(* CODESYS project cy-09-ifm-022_003.project
   Title: cy-09-ifm
   Author: AR
   Company: Clevergy S.r.l

Project tree, tasks and I/O mapping:
  Device : AC14nn, ifm electronic, order no. AC14nn, version 3.5.3.002
    application Application
      libraries: Standard, 3.5.5.0 (System); ACnnnn_Utils, * (ifm electronic); Util, 3.5.1.0 (System); SysRtc23, 3.4.0.0 (System); SysSocket23, 3.5.4.10 (System); SysFile, 3.5.6.0 (System); SysTypes Interfaces, * (System); CmpErrors Interfaces, * (System); VisuDialogs, * (System); NETWORK, 1.2.1.0 (OSCAT)
      task MainTask (cyclic, interval t#20ms, priority 15) calls PLC_PRG
      task EventTask (cyclic, interval t#20ms, priority 5) calls PLC_RT
      task VISU_TASK (cyclic, interval 100 ms, priority 30) calls VisuElems.Visu_Prg
      visualisation VIS_CHONOEDITOR
      visualisation PLC_VISU
    ASi_Master_1 : ASi Master 1, ifm electronic, version 3.5.3.002
      ASi_1_binaryIO : ASi_1_binaryIO, ifm ecomatic gmbh, version 3.5.3.002
          input  PSG01_IN : BOOL  // ASi Input bin.Digital S(A) Slave.Digital S(A) Slave[1].Bit0
          input  PSG02_IN : BOOL  // ASi Input bin.Digital S(A) Slave.Digital S(A) Slave[1].Bit2
          input  EXT_KEY1 : BOOL  // ASi Input bin.Digital S(A) Slave.Digital S(A) Slave[1].Bit3
          input  PSG03_IN : BOOL  // ASi Input bin.Digital S(A) Slave.Digital S(A) Slave[2].Bit0
          input  PSG04_IN : BOOL  // ASi Input bin.Digital S(A) Slave.Digital S(A) Slave[2].Bit2
          input  PSG05_IN : BOOL  // ASi Input bin.Digital S(A) Slave.Digital S(A) Slave[3].Bit0
          input  PSG06_IN : BOOL  // ASi Input bin.Digital S(A) Slave.Digital S(A) Slave[3].Bit2
          input  PSG07_IN : BOOL  // ASi Input bin.Digital S(A) Slave.Digital S(A) Slave[4].Bit0
          input  PSG08_IN : BOOL  // ASi Input bin.Digital S(A) Slave.Digital S(A) Slave[4].Bit2
          input  PSG09_IN : BOOL  // ASi Input bin.Digital S(A) Slave.Digital S(A) Slave[5].Bit0
          input  PSG10_IN : BOOL  // ASi Input bin.Digital S(A) Slave.Digital S(A) Slave[5].Bit2
          input  EXT_KEY2 : BOOL  // ASi Input bin.Digital S(A) Slave.Digital S(A) Slave[5].Bit3
          input  PSG11_IN : BOOL  // ASi Input bin.Digital S(A) Slave.Digital S(A) Slave[6].Bit0
          input  PSG12_IN : BOOL  // ASi Input bin.Digital S(A) Slave.Digital S(A) Slave[6].Bit2
          input  PSG13_IN : BOOL  // ASi Input bin.Digital S(A) Slave.Digital S(A) Slave[7].Bit0
          input  EXT_KEY3 : BOOL  // ASi Input bin.Digital S(A) Slave.Digital S(A) Slave[7].Bit3
          input  PSG14_IN : BOOL  // ASi Input bin.Digital S(A) Slave.Digital S(A) Slave[8].Bit0
          input  PSG15_IN : BOOL  // ASi Input bin.Digital S(A) Slave.Digital S(A) Slave[8].Bit2
          input  PSG16_IN : BOOL  // ASi Input bin.Digital S(A) Slave.Digital S(A) Slave[9].Bit0
          input  PSG17_IN : BOOL  // ASi Input bin.Digital S(A) Slave.Digital S(A) Slave[9].Bit2
          unmapped channels: ASi Input bin, ASi Output bin
      ASi_1_analogIO : ASi_1_analogIO, ifm ecomatic gmbh, version 3.5.3.002
          unmapped channels: ASi Input, ASi Output
    ASi_Master_2 : ASi Master 2, ifm electronic, version 3.5.3.002
      ASi_2_binaryIO : ASi_2_binaryIO, ifm ecomatic gmbh, version 3.5.3.002
          input  PSG18_IN : BOOL  // ASi Input bin.Digital S(A) Slave.Digital S(A) Slave[10].Bit0
          input  PSG19_IN : BOOL  // ASi Input bin.Digital S(A) Slave.Digital S(A) Slave[10].Bit2
          input  PSG20_IN : BOOL  // ASi Input bin.Digital S(A) Slave.Digital S(A) Slave[11].Bit0
          input  PSG21_IN : BOOL  // ASi Input bin.Digital S(A) Slave.Digital S(A) Slave[11].Bit1
          input  PSG22_IN : BOOL  // ASi Input bin.Digital S(A) Slave.Digital S(A) Slave[11].Bit2
          input  PSG23_IN : BOOL  // ASi Input bin.Digital S(A) Slave.Digital S(A) Slave[12].Bit0
          input  PSG24_IN : BOOL  // ASi Input bin.Digital S(A) Slave.Digital S(A) Slave[13].Bit0
          input  PSG25_IN : BOOL  // ASi Input bin.Digital S(A) Slave.Digital S(A) Slave[13].Bit1
          input  PSG26_IN : BOOL  // ASi Input bin.Digital S(A) Slave.Digital S(A) Slave[13].Bit2
          input  PSG27_IN : BOOL  // ASi Input bin.Digital S(A) Slave.Digital S(A) Slave[14].Bit0
          input  PSG28_IN : BOOL  // ASi Input bin.Digital S(A) Slave.Digital S(A) Slave[14].Bit1
          input  PSG29_IN : BOOL  // ASi Input bin.Digital S(A) Slave.Digital S(A) Slave[14].Bit2
          input  PSG30_IN : BOOL  // ASi Input bin.Digital S(A) Slave.Digital S(A) Slave[15].Bit0
          input  PSG31_IN : BOOL  // ASi Input bin.Digital S(A) Slave.Digital S(A) Slave[15].Bit1
          input  PSG32_IN : BOOL  // ASi Input bin.Digital S(A) Slave.Digital S(A) Slave[15].Bit2
          input  PSG33_IN : BOOL  // ASi Input bin.Digital S(A) Slave.Digital S(A) Slave[16].Bit0
          input  PSG34_IN : BOOL  // ASi Input bin.Digital S(A) Slave.Digital S(A) Slave[17].Bit0
          unmapped channels: ASi Input bin, ASi Output bin
      ASi_2_analogIO : ASi_2_analogIO, ifm ecomatic gmbh, version 3.5.3.002
          unmapped channels: ASi Input, ASi Output
    Fieldbus_Interface : Fieldbus Interface, ifm electronic, version 3.5.3.002
      FieldBusData_ : FieldBusData  , ifm ecomatic gmbh, version 3.5.3.002
          unmapped channels: Inputs from fieldbus, Outputs to fieldbus
      ASi_1_binaryOut : ASi_1_binaryOut, ifm ecomatic gmbh, version 3.5.3.002
          unmapped channels: FB ASi Output bin
      ASi_1_analogOut : ASi_1_analogOut, ifm ecomatic gmbh, version 3.5.3.002
          unmapped channels: FB ASi Output ana
      ASi_2_binaryOut : ASi_2_binaryOut, ifm ecomatic gmbh, version 3.5.3.002
          unmapped channels: FB ASi Output bin
      ASi_2_analogOut : ASi_2_analogOut, ifm ecomatic gmbh, version 3.5.3.002
          unmapped channels: FB ASi Output ana
    Ethernet : Ethernet, ifm electronic, version 3.4.2.0
        settings: IPAddress = [192,168,100,2]; SubnetMask = [255,255,255,0]; GatewayAddress = [0,0,0,0]
  POUs/
    Utils Functions/
      function ADDSTRING [ST]
      function block AVERAGE_DINT [ST]: Read, Reset
      function block AVERAGE_INT [ST]: Read, Reset
      function block AVERAGE_T [ST]: Read, Reset
      function CHKSTRING [ST]
      function COPY_32SWAP16 [ST]
      function DWORDSWAP [ST]
      function block FLT_EVENT [ST]
      function block FLT_TAP [ST]
      function block FLT_TIME [ST]
      function HEXTORAW [ST]
      function LINEAR [ST]
      function LINEAR_BAD [ST]
      function MEMCLR [ST]
      function MEMCPY [ST]
      function block DELAYRETRY [ST]: Start, Success, Fail
      function RAW16TOHEXSTR [ST]
      function RAWTOHEX [ST]
      function RAWTOHEXSTR [ST]
      function STR_NOSPACES [ST]
      function block TCPCLIENT [ST]
      function block TCPSERVER [ST]
      function block TONOF [ST]
      function ADR_AT_INT [ST]
    Utils/
      function CSV_Log [ST]
      function RTC_Update [ST]
    TCP_Logger/
      function LogEv [ST]
      function Logger_Head [ST]
      program Logger_Proc [ST]: MsgChk, MsgSave
      function Logger_Send [ST]
      function LogTrig [ST]
    Plant_Objects/
      function block obj_LUXM [ST]: AddLogData, StatReset
      function block obj_ZREL [ST]: AddLogData, MB_Req_NetStatus, MB_Set_DefaultMode, MB_Req_Status, MB_Set_AutoLearn, MB_Response
      function block obj_CRON [ST]: DB_Create, DB_Load, DB_SetName, Init, AddLogData
      function block obj_CRON_EDITOR [ST]: CA_Load_Exe, CA_Save_Exe, FileOpen, JL_Load_Exe, JL_Save_Exe, PR_Load_Exe, PR_Save_Exe
      function block obj_MODBUS_TCP [ST]: VARS_Process, VAR_Search
      function block obj_ASI [ST]
      function block obj_PSG [ST]: StatReset, AddLogData
      function block obj_ZGW [ST]: AddLogData
      function block obj_LICENSE [ST]
    program PLC_PRG [ST]: Main_Stm
    TCP_Remote/
      program Remote_Proc [ST]: Cmd_CAL, Cmd_CRON, Cmd_GRU, Cmd_PDC, Cmd_SYS, Command, Cmd_LUX
    Plant/
    program PLC_RT [ST]
    WagoLibModbus_IP_01/
      function block Client_OpenClose [ST]
      function block ETHERNET_MODBUSMASTER_TCP [ST]
      function Modbus_IP_Version [ST]
      function ModbusRequest [ST]
  _Datatypes/
    Logger/
      data type en_Logger_ErrLev
      data type en_Logger_Status
      data type typ_Logger
    data type en_SYS_Objects
    data type en_SYS_Status
    data type typ_SYS
    WagoLibModbus_IP_1/
      data type MODBUS_FC
    Plant_Objects/
      data type typ_Cron_Calendar
      data type typ_Cron_Jolly
      data type typ_Cron_Profile
      data type typ_MODBUS_VAR
  _Variables/
    global variables Global_Constants
    global variables Global_Retain
    global variables Global_Variables
  text list GlobalTextList
*)

// _Datatypes/Logger/en_Logger_ErrLev
TYPE en_Logger_ErrLev :
(
	EL_Log			:=0,
	EL_Wrn			:=1,
	EL_Alarm		:=2,
	EL_AlarmStop	:=3
);
END_TYPE

// _Datatypes/Logger/en_Logger_Status
TYPE en_Logger_Status :
(
	S_Logger_UNKNOWN := 0,
	S_Logger_IDLE,
	S_Logger_WAITCONN,
	S_Logger_WAITTX,
	S_Logger_WAITRESP,
	S_Logger_ERROR
);
END_TYPE

// _Datatypes/en_SYS_Objects
TYPE en_SYS_Objects :
(
	EO_SYS		:=0,  (* PLC *)
	EO_VPN		:=1,  (* VPN *)
	EO_DOOR		:=2,  (* Door & access control *)

	EO_CAL		:=10, (* Caldaia *)
	EO_CIR		:=11, (* Circolatore *)
	EO_CRON		:=12, (* Crono-termostato *)
	EO_VRD		:=13, (* Valvola miscelatore pannelli *)
	EO_CTL		:=14, (* Contalitri *)
	EO_CTB		:=15, (* Contabilizzatore *)
	EO_TPV		:=16, (* Temperature probes values *)
	EO_PPV		:=17, (* Pressure probes values *)
	EO_PBV		:=18, (* Over-Pressure Alarms *)
	EO_TBV		:=19, (* Over-Temperature Alarms *)
	EO_PMV		:=20, (* Under-Pressure Alarms *)
	EO_GRU		:=21, (* Gruppo termico *)
	EO_PDC		:=22, (* Pompa di calore *)
	EO_SOL		:=23, (* Pannello solare termico *)
	EO_ESOL		:=24, (* Pannello solare fotovoltaico *)
	EO_GAS		:=25, (* Contatore GAS *)
	EO_PORT		:=26, (* Misuratore di portata *)
	EO_FPV		:=27, (* Flow probes values *)
	EO_ANZ		:=28, (* Analizzatore di rete *)
	EO_SCA		:=29, (* Signal Control Alarms *)
	EO_LUX		:=30, (* Base Illumination point *)
	EO_LUXM		:=31, (* Metered Illumination point *)
	EO_PSG		:=32, (* Sensore di passaggio *)
	EO_HVAC		:=33, (* Heating, Ventilating and Air Conditioning *)
	EO_HYGRV	:=34, (* Relative Humidity sensors value *)
	EO_COOV		:=35, (* Carbon Dioxide CO2 sensors value *)

	EO_ZGW			:=200,  (* ZigBee - Gateway *)
	EO_ZRM			:=201,	(* ZigBee - Repeater *)
	EO_ZREL			:=202,	(* ZigBee - Actuator rele *)
	EO_ZTHL			:=203,	(* ZigBee - Temperature Sensor *)

	EO_ASGW			:=250,	(* ASi - Gateway *)
	EO_ASCBI		:=251,	(* ASi - Input Board, Ciabatta *)

	EO_LON			:=1000, (* Bus - LON *)
	EO_MODBUS		:=1001, (* Bus - MODBUS *)
	EO_MBUS			:=1002, (* Bus - M-BUS *)
	EO_MODBUS_TCP	:=1003, (* Bus - MODBUS TCP *)

	EO_GENERIC		:=9000, (* Generic dataset *)
	EO_EXPO			:=9001  (* EXPO dataset *)
);
END_TYPE

// _Datatypes/en_SYS_Status
TYPE en_SYS_Status :
(
	S_UNKNOWN  := 0,
	S_STARTUP,
	S_INIT_RTC,
	S_INIT_VAR,
	S_AUTOTEST,
	S_RUNNING,
	S_SHUTDOWN,
	S_HALT
);
END_TYPE

// _Datatypes/Logger/typ_Logger
TYPE typ_Logger :
STRUCT
	Status		: en_Logger_Status;

	SendReq		: BOOL;
	SendIdx		: DWORD;
	SendData	: ARRAY [0..MAX_SEND_TCP_CLIENT] OF BYTE;
	SendLen		: DINT;

	TData		: ARRAY [0..MAX_SEND_TCP_CLIENT] OF BYTE;
	TLen		: DINT;

	LastIdxPos	: DWORD;

	(* Temporary variables used by objects *)
	s1			: STRING(256);
	i1			: WORD;

END_STRUCT
END_TYPE

// _Datatypes/typ_SYS
TYPE typ_SYS :
STRUCT
	Status			: en_SYS_Status;
	Warning			: BOOL;
	Alarm			: BOOL;
	AlarmStop		: BOOL;

	Time_LogString	: STRING;
	Time_Year		: WORD;
	Time_Month		: BYTE;
	Time_Day		: BYTE;

	Time_CT_DT		: DT;
	Time_CT_Day		: WORD;
	Time_CT_Quarter	: BYTE;

	LastLogs_Idx	: BYTE;
	LastLogs_Dat	: ARRAY[0..5] OF STRING;
	LastLogs_Msg	: ARRAY[0..5] OF STRING;

END_STRUCT
END_TYPE

// _Datatypes/Plant_Objects/typ_Cron_Calendar
TYPE typ_Cron_Calendar :
STRUCT
	Profile		: ARRAY[0..384] OF BYTE;
END_STRUCT
END_TYPE

// _Datatypes/Plant_Objects/typ_Cron_Jolly
TYPE typ_Cron_Jolly :
STRUCT
	Start		: DT;
	End			: DT;
	Temp		: INT;
	Flags		: WORD; (* B0:Enabled B1..B15:Unused *)
END_STRUCT
END_TYPE

// _Datatypes/Plant_Objects/typ_Cron_Profile
TYPE typ_Cron_Profile :
STRUCT
	Flags		: WORD;
	Setpoint	: ARRAY [0..95] OF INT;
END_STRUCT
END_TYPE

// _Datatypes/Plant_Objects/typ_MODBUS_VAR
TYPE typ_MODBUS_VAR : (* Gestione parametri MODBUS *)
STRUCT
	SlaveAddress	: BYTE;
	FunCode			: BYTE;
	FunAddress		: WORD;
	Refresh_Time	: BYTE; (* 0:No refresh, x:Refresh in seconds *)
	Refresh_Cnt		: BYTE; (* -- INTERNAL do not use! -- *)
	Variable		: POINTER TO ARRAY[0..99] OF WORD;
	Variable_Size	: WORD; (* 1-100:Standard reading, 1001-1100:Swap32 *)
	Variable_Mirror : WORD; (* CHECKSUM - INTERNAL [Force refresh on read variables when <>0] *)
END_STRUCT
END_TYPE

// _Datatypes/WagoLibModbus_IP_1/MODBUS_FC
TYPE MODBUS_FC : (
	(*
	 * Class 0
 	*)
	READ_MULTIPLE_REGISTERS		:=16#03,
	WRITE_MULTIPLE_REGISTERS	:=16#10,
	(*
	 * Class 1
	 *)
	READ_COILS					:=16#01,
	READ_INPUT_DISCRETES		:=16#02,
	READ_INPUT_REGISTERS		:=16#04,
	WRITE_COIL					:=16#05,
	WRITE_SINGLE_REGISTER		:=16#06,
	READ_EXCEPTION_STATUS		:=16#07,
	(*
	 * Class 2
	 *)
	FORCE_MULTIPLE_COILS		:=16#0F,
	READ_WRITE_REGISTERS		:=16#17,

	(*
	 * Class ??
	 *)
	WRITE_MASK_REGISTER			:=16#16 (* 02.04.2013 UU *)

	);
END_TYPE

// _Variables/Global_Constants
{attribute 'global_init_slot' := '300'}
VAR_GLOBAL CONSTANT

	PSG_MAX	 : BYTE := 34;
	ZREL_MAX : BYTE := 38;
	CRON_MAX : BYTE := 38;
	LUXM_MAX : BYTE := 38;
	ACTIVELUX: BYTE := 17;

	(* Filesystem *)
	LogsPath			: STRING :='/media/sd/';
	ConfPath			: STRING :='/media/sd/';
	//FilesPath			: STRING :='/media/sd/';(*'';*)(*'S:\';*)

	(* Visu colours *)	
	COLOR_RED 		: DWORD:=16#F02020;
	COLOR_YELLOW	: DWORD:=16#F0F020;
	COLOR_GREEN		: DWORD:=16#20F020;
	COLOR_GREEN_OFF : DWORD:=16#108010;
	COLOR_LBLUE		: DWORD:=16#80F0F0;
	COLOR_GREY		: DWORD:=16#C0C0C0;
	
	(******************************************************)
	(**************** MOVE OUTSIDE HERE *******************)
	(* TCP Logger *)
	Logger_SERVER		: STRING:='';
	Logger_IP			: STRING:='192.168.100.3'; //'192.168.100.3';   '178.33.227.41';
	Logger_PORT			: WORD  :=80;
	Logger_GETSTART		: STRING:='GET /cygmsrv/AFLgm.ashx?';
	Logger_GETEND		: STRING:='$R$N$R$N';
	Logger_CHECK		: STRING:='True';
	Logger_CRLF			: STRING:='$R$N';
	Logger_DataFile		: STRING:='LOG.DAT';
	Logger_DataFileOld	: STRING:='LOG.BCK';
	Logger_IndexFile	: STRING:='LOG.IDX';
	Logger_ConnRetries	: BYTE:=5;
	Logger_RecoverMsgs	: BYTE:=50;
	(* TCP Remote *)
	Remote_PORT			: WORD  :=10;
	Remote_WELCOME		: STRING:='Connected$R$N';
	(* TCP Sockets *)
	MAX_SEND_TCP_SERVER					 : DWORD:=1500;(*60000*)
	MAX_RECEIVE_TCP_SERVER				 : WORD:=3000;	//DWORD:=3000; GIURE ver 22_001
	MAX_RECEIVE_TCP_SERVER_SOCKET	 	 : DWORD:=1500;
	MAX_SEND_TCP_CLIENT					 : DWORD:=4096;(*15000*)
	MAX_RECEIVE_TCP_CLIENT				 : DWORD:=1500;
	MAX_RECEIVE_TCP_CLIENT_SOCKET		 : DWORD:=1500;
	MAX_RECEIVE_UDP_SERVER				 : INT  :=1472;
	MAX_RECEIVE_UDP_CLIENT				 : INT  :=1472;
	CONNECT_WATCHDOG_TIME				 : TIME :=T#10S;
	(******************************************************)

END_VAR

// _Variables/Global_Retain
VAR_GLOBAL RETAIN
	Mode_Manual : BOOL := FALSE;

	PASSAGES		: ARRAY [1..PSG_MAX] OF DWORD;

	WORKINGTIME		: ARRAY [1..LUXM_MAX] OF DWORD; (* [sec] Internal working time counter *)
	POWERONCYCLES	: ARRAY [1..LUXM_MAX] OF DWORD; (* Internal counter of power-on cycles *)
	ENERGYCOUNTER	: ARRAY [1..LUXM_MAX] OF DWORD; (* [E-1 kWh] Internal energy counter *)
	ENERGYCOUNTER_T : ARRAY [1..LUXM_MAX] OF DWORD; (* Temporary energy in E-2*Wsec *)
	
	LicenseManager:obj_LICENSE;

END_VAR

// _Variables/Global_Variables
VAR_GLOBAL
	Plant_NAME			: STRING :='cySN:9 cyVER:18 - AF-Logistics Bazar';	//'cySN:9 cyVER:18 - AF-Logistics Bazar';	
	Plant_SN			: DWORD  :=9;	//:=9; 	(* S/N Impianto di telecontrollo *)
	Plant_SW_VER		: WORD   :=18;		(* Versione SW installata *)

	SYS    : typ_SYS;
	Logger : typ_Logger;
	CronEd : obj_CRON_EDITOR;

	(**** PLANT OBJECTS ****)
	ASI01: obj_ASI				:=( ID:=1 );
	ASI02: obj_ASI				:=( ID:=2 );

	PSG		: ARRAY [1..PSG_MAX] OF obj_PSG;
	
	MODB01 : obj_MODBUS_TCP		:= ( ID:=1, IP:='192.168.100.4');	//'192.168.100.4' ); '10.186.79.9'
	ZGW01  : obj_ZGW			:= ( ID:=1, ADDRESS:=99  );

	ZREL   : ARRAY [1..ZREL_MAX] OF obj_ZREL;
	CRON   : ARRAY [1..CRON_MAX] OF obj_CRON;
	LUXM   : ARRAY [1..LUXM_MAX] OF obj_LUXM;
	
	ZREL_STATUS_ALIGNED   : ARRAY [1..ZREL_MAX] OF BOOL;

	(**** SIMULATION ONLY ****)
	TEST1:BOOL;	
	KEYON:BOOL;
	KEYVIRT:BOOL;
	(*...*)
	
	testCronoOn:BOOL:=FALSE;
	testCronoOff:BOOL:=FALSE;

END_VAR

// POUs/PLC_PRG
PROGRAM PLC_PRG
VAR
	Timer1	: TON; (* Fast controls tick *)
	Timer2	: TON; (* Plant control tick *)
	Timer3	: TON; (* Logger timer *)
	i 		: BYTE;
	ValInCrono	:	INT; //Valore del setpoint del crono
	LuxSelected	:	INT;//lux selezionato in plc visu per on/off
	TimerLuxSelected	:	INT;//lux selezionato in plc visu per modifica timer
	//ListaLux 	:	ARRAY [ACTIVELUX..LUXM_MAX] OF BOOL; 
	
END_VAR

(******************************************************************************
 ****                           MAIN TASK CODE                             ****
 ******************************************************************************

	Network setup:
		IP  = 192.168.100.2 | MSK = 255.255.255.0
		GW	= 192.168.100.1 | DNS = 192.168.100.1
		SNTP = 193.204.114.232 (3600s) ==> 192.168.100.3

*)

LicenseManager();

IF LicenseManager.IS_LICENSED THEN

(*==============================*)
(*===== Main status machine ====*)
(*==============================*)
Main_Stm();
Remote_Proc();		
(*==============================*)
(*== Running cycle operations ==*)
(*==============================*)

IF SYS.Status>S_INIT_VAR THEN
	(* Execute cycle processes *)
	MODB01();
	FOR i := 1 TO ACTIVELUX DO	//Cicla sulle lampade 1 - 17 controllate da fotocellula
		ZREL[i]( MODBUS:=MODB01, REL_CTRL:=LUXM[i].REL_EN );
	END_FOR
	FOR i := ACTIVELUX+1 TO LUXM_MAX DO //Cicla sulle lampade 18 - 38 controllate da crono
		ZREL[i]( MODBUS:=MODB01, REL_CTRL:=LUXM[i].REL_EN );
	END_FOR
END_IF

(*==============================*)
(*== System cycle operations ===*)
(*==============================*)
(* Execute TCP processes *)
Logger_Proc();
//Remote_Proc();		
(* Update user led *)
(*USRLED_Update();*)
(* Execute Cron Editor commands *)
CronEd();
(* External resources *)
(*
   IF NOT TPV01.ERR THEN T_AMB:=T_S01;
ELSIF NOT TPV05.ERR THEN T_AMB:=GRU01.TAmb;
ELSE 					 T_AMB:=Plant_DefaultTAmb;
END_IF
*)

(**** SIMULATION ONLY ****)
(*...*)

END_IF

ACTION Main_Stm:
CASE Sys.Status OF

	S_STARTUP:
		(* Initialize array objects *)
		FOR i := 1 TO PSG_MAX  DO PSG[i].ID:=i;  END_FOR
		FOR i := 1 TO ZREL_MAX DO ZREL[i].ID:=i; ZREL[i].ADDRESS:=i*2; ZREL[i].ADDRESSGW:=i*2-1; END_FOR
		FOR i := 1 TO CRON_MAX DO CRON[i].ID:=i; END_FOR
		FOR i := 1 TO LUXM_MAX DO LUXM[i].ID:=i; END_FOR
		FOR i := 1 TO ACTIVELUX DO LUXM[i].CTRL_MODE_backUp := LUXM[i].CTRL_MODE; END_FOR
		Sys.Status:=S_INIT_RTC;

	S_INIT_RTC:
		(* Check RTC and update from network *)
		RTC_Update();
		(* Check time *)
		IF Sys.Time_Year>2000 THEN
			Sys.Status:=S_INIT_VAR;
		END_IF

	S_INIT_VAR:
		LogEv(EL_Wrn,EO_SYS,0,1,CONCAT('System_startup_v',WORD_TO_STRING(Plant_SW_VER)));
		Sys.Status:=S_RUNNING;

	S_RUNNING:
		
		IF(testCronoOn) THEN
			LUXM[18].PressKeyVisuMan:=TRUE;
			LUXM[18].PressKeyVisuOn:=TRUE;

			LUXM[19].PressKeyVisuMan:=TRUE;
			LUXM[19].PressKeyVisuOn:=TRUE;

			LUXM[20].PressKeyVisuMan:=TRUE;
			LUXM[20].PressKeyVisuOn:=TRUE;

			LUXM[21].PressKeyVisuMan:=TRUE;
			LUXM[21].PressKeyVisuOn:=TRUE;

			LUXM[22].PressKeyVisuMan:=TRUE;
			LUXM[22].PressKeyVisuOn:=TRUE;

			LUXM[23].PressKeyVisuMan:=TRUE;
			LUXM[23].PressKeyVisuOn:=TRUE;

			LUXM[24].PressKeyVisuMan:=TRUE;
			LUXM[24].PressKeyVisuOn:=TRUE;

			LUXM[25].PressKeyVisuMan:=TRUE;
			LUXM[25].PressKeyVisuOn:=TRUE;

			LUXM[26].PressKeyVisuMan:=TRUE;
			LUXM[26].PressKeyVisuOn:=TRUE;

			LUXM[27].PressKeyVisuMan:=TRUE;
			LUXM[27].PressKeyVisuOn:=TRUE;

			LUXM[28].PressKeyVisuMan:=TRUE;
			LUXM[28].PressKeyVisuOn:=TRUE;

			LUXM[29].PressKeyVisuMan:=TRUE;
			LUXM[29].PressKeyVisuOn:=TRUE;

			LUXM[30].PressKeyVisuMan:=TRUE;
			LUXM[30].PressKeyVisuOn:=TRUE;

			LUXM[31].PressKeyVisuMan:=TRUE;
			LUXM[31].PressKeyVisuOn:=TRUE;

			LUXM[32].PressKeyVisuMan:=TRUE;
			LUXM[32].PressKeyVisuOn:=TRUE;

			LUXM[33].PressKeyVisuMan:=TRUE;
			LUXM[33].PressKeyVisuOn:=TRUE;

			LUXM[34].PressKeyVisuMan:=TRUE;
			LUXM[34].PressKeyVisuOn:=TRUE;

			LUXM[35].PressKeyVisuMan:=TRUE;
			LUXM[35].PressKeyVisuOn:=TRUE;

			LUXM[36].PressKeyVisuMan:=TRUE;
			LUXM[36].PressKeyVisuOn:=TRUE;

			LUXM[37].PressKeyVisuMan:=TRUE;
			LUXM[37].PressKeyVisuOn:=TRUE;

			LUXM[38].PressKeyVisuMan:=TRUE;
			LUXM[38].PressKeyVisuOn:=TRUE;

		
			testCronoOn:=FALSE;
	
		END_IF
		
		IF(testCronoOff) THEN
			LUXM[18].PressKeyVisuMan:=TRUE;
			LUXM[18].PressKeyVisuOn:=FALSE;

			LUXM[19].PressKeyVisuMan:=TRUE;
			LUXM[19].PressKeyVisuOn:=FALSE;

			LUXM[20].PressKeyVisuMan:=TRUE;
			LUXM[20].PressKeyVisuOn:=FALSE;

			LUXM[21].PressKeyVisuMan:=TRUE;
			LUXM[21].PressKeyVisuOn:=FALSE;

			LUXM[22].PressKeyVisuMan:=TRUE;
			LUXM[22].PressKeyVisuOn:=FALSE;

			LUXM[23].PressKeyVisuMan:=TRUE;
			LUXM[23].PressKeyVisuOn:=FALSE;

			LUXM[24].PressKeyVisuMan:=TRUE;
			LUXM[24].PressKeyVisuOn:=FALSE;

			LUXM[25].PressKeyVisuMan:=TRUE;
			LUXM[25].PressKeyVisuOn:=FALSE;

			LUXM[26].PressKeyVisuMan:=TRUE;
			LUXM[26].PressKeyVisuOn:=FALSE;

			LUXM[27].PressKeyVisuMan:=TRUE;
			LUXM[27].PressKeyVisuOn:=FALSE;

			LUXM[28].PressKeyVisuMan:=TRUE;
			LUXM[28].PressKeyVisuOn:=FALSE;

			LUXM[29].PressKeyVisuMan:=TRUE;
			LUXM[29].PressKeyVisuOn:=FALSE;

			LUXM[30].PressKeyVisuMan:=TRUE;
			LUXM[30].PressKeyVisuOn:=FALSE;

			LUXM[31].PressKeyVisuMan:=TRUE;
			LUXM[31].PressKeyVisuOn:=FALSE;

			LUXM[32].PressKeyVisuMan:=TRUE;
			LUXM[32].PressKeyVisuOn:=FALSE;

			LUXM[33].PressKeyVisuMan:=TRUE;
			LUXM[33].PressKeyVisuOn:=FALSE;

			LUXM[34].PressKeyVisuMan:=TRUE;
			LUXM[34].PressKeyVisuOn:=FALSE;

			LUXM[35].PressKeyVisuMan:=TRUE;
			LUXM[35].PressKeyVisuOn:=FALSE;

			LUXM[36].PressKeyVisuMan:=TRUE;
			LUXM[36].PressKeyVisuOn:=FALSE;

			LUXM[37].PressKeyVisuMan:=TRUE;
			LUXM[37].PressKeyVisuOn:=FALSE;

			LUXM[38].PressKeyVisuMan:=TRUE;
			LUXM[38].PressKeyVisuOn:=FALSE;

		
			testCronoOff:=FALSE;
	
		END_IF
		
		Timer1(IN:=NOT Timer1.Q,PT:=T#50ms);
		IF Timer1.Q THEN
			(* Update meters *)

			(* Update system checks *)
			//SYS_Proc();
			//SCA_Proc();
		END_IF

		Timer2(IN:=NOT Timer2.Q,PT:=T#500ms);
		IF Timer2.Q THEN
			(* Read current date/time *)
			RTC_Update();
			(* Sensors assignment *)
			LUXM[ 1].CTRL_TRIG:=PSG[ 1].SENSE_TRIG OR PSG[30].SENSE_TRIG;
			LUXM[ 2].CTRL_TRIG:=PSG[ 2].SENSE_TRIG OR PSG[30].SENSE_TRIG OR PSG[31].SENSE_TRIG;
			LUXM[ 3].CTRL_TRIG:=PSG[ 3].SENSE_TRIG OR PSG[32].SENSE_TRIG OR PSG[31].SENSE_TRIG;
			LUXM[ 4].CTRL_TRIG:=PSG[ 4].SENSE_TRIG OR PSG[32].SENSE_TRIG OR PSG[27].SENSE_TRIG;
			LUXM[ 5].CTRL_TRIG:=PSG[ 5].SENSE_TRIG OR PSG[28].SENSE_TRIG OR PSG[27].SENSE_TRIG;
			LUXM[ 6].CTRL_TRIG:=PSG[ 6].SENSE_TRIG OR PSG[28].SENSE_TRIG OR PSG[29].SENSE_TRIG;
			LUXM[ 7].CTRL_TRIG:=PSG[ 7].SENSE_TRIG OR PSG[24].SENSE_TRIG OR PSG[29].SENSE_TRIG;
			LUXM[ 8].CTRL_TRIG:=PSG[ 8].SENSE_TRIG OR PSG[24].SENSE_TRIG OR PSG[25].SENSE_TRIG;
			LUXM[ 9].CTRL_TRIG:=PSG[ 9].SENSE_TRIG OR PSG[26].SENSE_TRIG OR PSG[25].SENSE_TRIG;
			LUXM[10].CTRL_TRIG:=PSG[10].SENSE_TRIG OR PSG[26].SENSE_TRIG OR PSG[23].SENSE_TRIG;
			LUXM[11].CTRL_TRIG:=PSG[11].SENSE_TRIG OR PSG[33].SENSE_TRIG OR PSG[23].SENSE_TRIG;
			LUXM[12].CTRL_TRIG:=PSG[12].SENSE_TRIG OR PSG[33].SENSE_TRIG OR PSG[34].SENSE_TRIG; 
			LUXM[13].CTRL_TRIG:=PSG[13].SENSE_TRIG OR PSG[20].SENSE_TRIG OR PSG[34].SENSE_TRIG;
			LUXM[14].CTRL_TRIG:=PSG[14].SENSE_TRIG OR PSG[20].SENSE_TRIG OR PSG[21].SENSE_TRIG;
			LUXM[15].CTRL_TRIG:=PSG[15].SENSE_TRIG OR PSG[22].SENSE_TRIG OR PSG[21].SENSE_TRIG;
			LUXM[16].CTRL_TRIG:=PSG[16].SENSE_TRIG OR PSG[22].SENSE_TRIG OR PSG[18].SENSE_TRIG;
			LUXM[17].CTRL_TRIG:=PSG[17].SENSE_TRIG OR PSG[19].SENSE_TRIG OR PSG[18].SENSE_TRIG;
			(* External switch *)
			KEYON:=EXT_KEY1 OR EXT_KEY2 OR EXT_KEY3 OR KEYVIRT;
			(* Clear sensors trigger *)
			FOR i :=1 TO PSG_MAX DO PSG[i].SENSE_TRIG:=FALSE; END_FOR
			(* Execute plant operations *)
			FOR i := 1 TO ACTIVELUX DO //Set delle lampade 1-17 a controllo con fotocellule e lettura degli stati dei relè
				if (( LUXM[i].PressKeyVisuMan = FALSE) and ( LUXM[i].TCP_CommandMAN = FALSE))then //se non ci sono comandi manuali da visu o da tcp
					LUXM[i].ModeToServer := 3;  // Mode per log per lux a Timer soggetto a passaggi
					LUXM[i].CTRL_MODE:=LUXM[i].CTRL_MODE_backUp;
				else if (( LUXM[i].PressKeyVisuOn) and ( LUXM[i].PressKeyVisuMan)) or (( LUXM[i].TCP_CommandMAN) and ( LUXM[i].TCP_CommandON)) then //se ci sono comandi manuali e ON
						LUXM[i].ModeToServer := 1;  // Mode per log per lux in manuale ON 	
						LUXM[i].CTRL_MODE:=-1;
					else 
						if (( LUXM[i].PressKeyVisuOn = FALSE) and ( LUXM[i].PressKeyVisuMan)) or (( LUXM[i].TCP_CommandMAN) and ( LUXM[i].TCP_CommandON = FALSE)) then //se ci sono comandi manuali e OFF
							LUXM[i].ModeToServer := 0;  // Mode per log per lux in manuale ON 	
							LUXM[i].CTRL_MODE:=0;	
						end_if				
					end_if
				end_if
				LUXM[i]( WORKINGTIME:=WORKINGTIME[i],     POWERONCYCLES:=POWERONCYCLES[i],
						 ENERGYCOUNTER:=ENERGYCOUNTER[i], ENERGYCOUNTER_T:=ENERGYCOUNTER_T[i],
						 CTRL_EXTON:=KEYON );
				(* Copy sensitive states to loads *)
				LUXM[i].REL_ST :=ZREL[i].REL_ST;
				LUXM[i].REL_V  :=ZREL[i].REL_V;
				LUXM[i].REL_A  :=ZREL[i].REL_A;
				LUXM[i].REL_ALM:=ZREL[i].REL_ALM;
			END_FOR
			
			FOR i := ACTIVELUX+1 TO LUXM_MAX DO //Set delle lampade 18-38 a controllo con crono e lettura degli stati dei relè
				LUXM[i].ModeToServer := 2;  // Mode per log per lux a Crono 
				CRON[i]( SETPOINT=>ValInCrono );
				if (( LUXM[i].PressKeyVisuMan = FALSE) and ( LUXM[i].TCP_CommandMAN = FALSE))then //se non ci sono comandi manuali da visu o da tcp
					if ValInCrono = 1000 then
						LUXM[i].CTRL_MODE:=-1;
					elsif  ValInCrono = 0 then
						LUXM[i].CTRL_MODE:=0;
					end_if
				else if (( LUXM[i].PressKeyVisuOn) and ( LUXM[i].PressKeyVisuMan)) or (( LUXM[i].TCP_CommandMAN) and ( LUXM[i].TCP_CommandON)) then //se ci sono comandi manuali e ON
						LUXM[i].ModeToServer := 1;  // Mode per log per lux in manuale ON 	
						LUXM[i].CTRL_MODE:=-1;
					else 
						if (( LUXM[i].PressKeyVisuOn = FALSE) and ( LUXM[i].PressKeyVisuMan)) or (( LUXM[i].TCP_CommandMAN) and ( LUXM[i].TCP_CommandON = FALSE)) then //se ci sono comandi manuali e OFF
							LUXM[i].ModeToServer := 0;  // Mode per log per lux in manuale ON 	
							LUXM[i].CTRL_MODE:=0;	
						end_if				
					end_if
				end_if
(*				IF ValInCrono = 1000 OR (( LUXM[i].PressKeyVisuOn) and ( LUXM[i].PressKeyVisuMan)) or ( LUXM[i].TCP_Command = 1)//LuxSelected = i AND
					THEN
						if (( LUXM[i].PressKeyVisuOn) and ( LUXM[i].PressKeyVisuMan)) or ( LUXM[i].TCP_Command = 1) then
							LUXM[i].ModeToServer := 1;  // Mode per log per lux in manuale ON 			
						end_if
						LUXM[i].CTRL_MODE:=-1;
					ELSE IF ValInCrono = 0 OR (( Not LUXM[i].PressKeyVisuOn) and ( LUXM[i].PressKeyVisuMan)) or ( LUXM[i].TCP_Command = 0) //LuxSelected = i AND
						THEN
							if (( Not LUXM[i].PressKeyVisuOn) and ( LUXM[i].PressKeyVisuMan))  or ( LUXM[i].TCP_Command = 0) then
								LUXM[i].ModeToServer := 0;  // Mode per log per lux in manuale OFF 	
							end_if
							LUXM[i].CTRL_MODE:=0;	
					END_IF
				END_IF
				*)
				(*LUXM[i].CTRL_MODE:=CRON[i].SetPoint;*)
				LUXM[i]( WORKINGTIME:=WORKINGTIME[i],     POWERONCYCLES:=POWERONCYCLES[i],
						 ENERGYCOUNTER:=ENERGYCOUNTER[i], ENERGYCOUNTER_T:=ENERGYCOUNTER_T[i],
						 CTRL_EXTON:=KEYON );
				(* Copy sensitive states to loads *)
				LUXM[i].REL_ST :=ZREL[i].REL_ST;
				LUXM[i].REL_V  :=ZREL[i].REL_V;
				LUXM[i].REL_A  :=ZREL[i].REL_A;
				LUXM[i].REL_ALM:=ZREL[i].REL_ALM;
			END_FOR
			(* ASi Diagnostics *)
			ASI01();
			ASI02();
			(* Test toggle *)
			IF TEST1 THEN TEST1:=FALSE; ELSE TEST1:=TRUE; END_IF
		END_IF

		Timer3(IN:=NOT Timer3.Q,PT:=T#5m);
		IF Timer3.Q THEN
			(* Trig logger *)
			LogTrig();
			(* Execute temporary CSV logger *)
			(*CSV_Log();*)
		END_IF

	S_SHUTDOWN:
		(* Stop sistema *)
		Sys.Status:=S_STARTUP;

	S_HALT:
		(* Aspetta uscita manuale *)
		Sys.Status:=S_STARTUP;

ELSE
	Sys.Status:=S_STARTUP;
END_CASE;
END_ACTION

END_PROGRAM

// POUs/TCP_Remote/Remote_Proc
PROGRAM Remote_Proc
VAR
	s1:         	TCPSERVER;
	Enable: 		BOOL;
	Connected: 		BOOL;
	Error: 			DINT;

	TxData:			ARRAY [0..MAX_SEND_TCP_SERVER] OF BYTE;
	TxLen:			DINT;
	TxTrig:			BOOL;

	RxData:			ARRAY [0..MAX_RECEIVE_TCP_SERVER] OF BYTE;
	RxLen:			DINT;

	Status:			DINT;

	(* Command interpreter *)

	Cmd_Buf:		ARRAY [0..MAX_RECEIVE_TCP_SERVER] OF BYTE;
	Cmd_Buf_U16:	POINTER TO WORD;
	Cmd_Buf_INT:	POINTER TO INT;
	Cmd_BufLen:		WORD;
	Cmd_St:			WORD;

	Cmd_Obj:		en_SYS_Objects;	// GIURE ver 206 WORD;
	Cmd_ObjIdx:		WORD;
	Cmd_C:			WORD;
	Cmd_R:			WORD;
	Cmd_CLen:		WORD;
	Cmd_RLen:		WORD;

	i : WORD;
	j : INT;
	s2 : STRING;
	x : word;
	NewValueTimer: dword;	
	
	Result: bool;
	DateTime: DT;
	DTStr: string;
	Year: word;
	Month, Day, Hour, minute, Sec: byte;
	LocalSetpoint: array[0..95] of word;
	Plant_SN_H_W, Plant_SN_L_W:	word;
	Plant_SN_H, Plant_SN_L: dword;
	NewValueTimerH, NewValueTimerL: word;
	ModeFromPlc	: word;
END_VAR

(*=== State machine ===*)
CASE Status OF
	0: (* Startup *)
		TxLen:=0; TxTrig:=FALSE;
		RxLen:=0;
		Enable:=TRUE;
		Status:=1;

	1: (* Wait incoming connection *)
		IF Connected THEN
			(* Log access *)
			//LogEv(EL_Log,EO_VPN,1,5,'Remote');
			(* Send welcome message *)
			(*ADDSTRING(pTxData:=ADR(TxData), pString:=ADR(Remote_WELCOME), TxLen:=TxLen);
			TxTrig:=TRUE;*)
			(* Reset vars *)
			Cmd_BufLen:=0;
			Cmd_St:=0;
			Status:=2;
		END_IF
		IF Error>1 THEN
			Enable:=FALSE;
			Status:=0;
		END_IF

	2: (* Wait command *)
		IF RxLen>0 THEN
			(*=== Interpreter start ===*)
			IF Cmd_BufLen+(RxLen/2)>=MAX_RECEIVE_TCP_SERVER THEN
				(* ERROR *)
				Cmd_BufLen:=0;
			ELSE
				i:=HEXTORAW(pString:=ADR(RxData), StringLen:=DINT_TO_WORD(RxLen), pData:=ADR(Cmd_Buf[Cmd_BufLen]));
				Cmd_BufLen:=Cmd_BufLen+i;
			END_IF
			IF Cmd_BufLen>=8 THEN
				Cmd_Buf_U16:=ADR(Cmd_Buf[6]);
//				IF Cmd_BufLen>=(8+Cmd_Buf_U16^) THEN
//					Cmd_CLen:=Cmd_Buf_U16^;
//					Cmd_Buf_U16:=ADR(Cmd_Buf[0]); Cmd_Obj:=Cmd_Buf_U16^;
//					Cmd_Buf_U16:=ADR(Cmd_Buf[2]); Cmd_ObjIdx:=Cmd_Buf_U16^;
//					Cmd_Buf_U16:=ADR(Cmd_Buf[4]); Cmd_C:=Cmd_Buf_U16^;
				IF Cmd_BufLen>=(8+byte_to_word(Cmd_Buf[6])) THEN	
					Cmd_Obj:=byte_to_word(Cmd_Buf[0]);
					Cmd_ObjIdx:=byte_to_word(Cmd_Buf[3]); //memorizzo il byte più significativo (yy) di |xxyy|
					Cmd_ObjIdx:=SHL(Cmd_ObjIdx,8); //shift a sx di 8 bit
					Cmd_ObjIdx:=Cmd_ObjIdx+byte_to_word(Cmd_Buf[2]); //aggiungo il byte meno significativo (xx)
					Cmd_C:=byte_to_word(Cmd_Buf[4]);
					Cmd_CLen:=byte_to_word(Cmd_Buf[6]);
					(* Log command *)
					(*
					s2:='RCmd_';		s2:=CONCAT(s2,WORD_TO_STRING(Cmd_Obj));
					s2:=CONCAT(s2,'_'); s2:=CONCAT(s2,WORD_TO_STRING(Cmd_ObjIdx));
					s2:=CONCAT(s2,'_'); s2:=CONCAT(s2,WORD_TO_STRING(Cmd_C));
					s2:=CONCAT(s2,'_');	s2:=CONCAT(s2,WORD_TO_STRING(Cmd_CLen));
					LogEv(EL_Log,EO_VPN,1,6,s2);
					*)
					(* Execute command *)
					Command();
					Cmd_BufLen:=0;
				END_IF
			END_IF
			(*=== Interpreter end ===*)
			RxLen:=0;
		END_IF
		IF NOT Connected THEN
			Status:=0;
		END_IF

ELSE
	Status:=0;
END_CASE


(*=== Execute server lib ===*)
s1(
	xEnable				:= Enable,
	wPortNumber			:= Remote_PORT,
	tServerTimeOut		:= t#10s,//t#15m,
	ptSendData			:= ADR(TxData),
	diSendCount			:= TxLen,
	xStartSend			:= TxTrig,
	aReceiveBuffer		:= RxData,
	diReceiveCount		:= RxLen,
	xClientConnected	=> Connected,
	diError				=> Error
);

ACTION Cmd_CAL:
(* Check index *)
IF Cmd_ObjIdx<1 OR Cmd_ObjIdx>17 THEN
	Cmd_R:=2;
	RETURN;
END_IF

(* Process command *)
CASE Cmd_C OF

	1: (* TRY REARM *)

	
ELSE
	Cmd_R:=3;
END_CASE
END_ACTION

ACTION Cmd_CRON:
(* Check index *)
//IF Cmd_ObjIdx<1 OR Cmd_ObjIdx>38 THEN 
IF Cmd_ObjIdx<=ACTIVELUX OR Cmd_ObjIdx>LUXM_MAX THEN	//eseguo controllo che siano i lux a crono e non a timer su passaggio
	Cmd_R:=2;
	RETURN;
END_IF

(* Process command *)
CASE Cmd_C OF

	1: (* GET PROFILE *)
		IF Cmd_CLen<>3 THEN
			Cmd_R:=4;
		ELSE
			(* Load profile *)
			CronEd.CN_Sel:=WORD_TO_BYTE(Cmd_ObjIdx);
			CronEd.CN_YSel:=Cmd_Buf[9];					//**
			CronEd.CN_YSel:=shl(CronEd.CN_YSel, 8);		//**
			CronEd.CN_YSel:=CronEd.CN_YSel+Cmd_Buf[8];	//**
//			Cmd_Buf_U16:=ADR(Cmd_Buf[8]); Sostituisco questa riga e la seguente con le 3 precedenti per little/big endian (**)
//			CronEd.CN_YSel:=Cmd_Buf_U16^;
			CronEd.PR_Sel:=Cmd_Buf[10];
			CronEd.PR_Load_Exe();
			for x:=0 to 95 do
				LocalSetpoint[x]:= int_to_word(CronEd.PR.Setpoint[x]);
				LocalSetpoint[x]:=rol(LocalSetpoint[x], 8); //Scambio byte per compatibilità con sistema wago little endian
			end_for
			(* Copy data *)
			Cmd_RLen:=192;
//			TxLen:=TxLen+RAWTOHEX(ADR(CronEd.PR.Setpoint),192,ADR(TxData[TxLen]));
			TxLen:=TxLen+RAWTOHEX(ADR(LocalSetpoint),192,ADR(TxData[TxLen]));
		END_IF

	2: (* SET PROFILE *)
		IF Cmd_CLen<>(3+192) THEN
			Cmd_R:=4;
		ELSE
			(* Save profile *)
			CronEd.CN_Sel:=WORD_TO_BYTE(Cmd_ObjIdx);
			CronEd.CN_YSel:=Cmd_Buf[9];					//**
			CronEd.CN_YSel:=shl(CronEd.CN_YSel, 8);		//**
			CronEd.CN_YSel:=CronEd.CN_YSel+Cmd_Buf[8];	//**
//			Cmd_Buf_U16:=ADR(Cmd_Buf[8]); Sostituisco questa riga e la seguente con le 3 precedenti per little/big endian (**)
//			CronEd.CN_YSel:=Cmd_Buf_U16^;
			CronEd.PR_Sel:=Cmd_Buf[10];
			MEMCPY(ADR(Cmd_Buf[11]),ADR(LocalSetpoint),192); //copio i dati in locale
			for x:=0 to 95 do
				LocalSetpoint[x]:=rol(LocalSetpoint[x], 8); //Scambio byte per compatibilità con sistema wago little endian
			end_for
			MEMCPY(ADR(LocalSetpoint),ADR(CronEd.PR.Setpoint),192); //copio i byte scambiati sopra nel setpoint del crono 
//			MEMCPY(ADR(Cmd_Buf[11]),ADR(CronEd.PR.Setpoint),192);
			CronEd.PR_Save_Exe();
		END_IF

	5: (* GET CALENDAR MONTH *)  
		IF Cmd_CLen<>3 THEN
			Cmd_R:=4;
		ELSE
			(* Load calendar *)
			CronEd.CN_Sel:=WORD_TO_BYTE(Cmd_ObjIdx);
			CronEd.CN_YSel:=Cmd_Buf[9];					//**
			CronEd.CN_YSel:=shl(CronEd.CN_YSel, 8);		//**
			CronEd.CN_YSel:=CronEd.CN_YSel+Cmd_Buf[8];	//**
//			Cmd_Buf_U16:=ADR(Cmd_Buf[8]); Sostituisco questa riga e la seguente con le 3 precedenti per little/big endian (**)
//			CronEd.CN_YSel:=Cmd_Buf_U16^;
			CronEd.CA_Sel:=Cmd_Buf[10];
			CronEd.CA_Load_Exe();
			(* Copy data *)
			Cmd_RLen:=32;
			TxLen:=TxLen+RAWTOHEX(ADR(CronEd.CA.Profile),32,ADR(TxData[TxLen]));
		END_IF

	6: (* SET CALENDAR MONTH *)	
		IF Cmd_CLen<>(3+32) THEN
			Cmd_R:=4;
		ELSE
			(* Save calendar *)
			CronEd.CN_Sel:=WORD_TO_BYTE(Cmd_ObjIdx);
			CronEd.CN_YSel:=Cmd_Buf[9];					//**
			CronEd.CN_YSel:=shl(CronEd.CN_YSel, 8);		//**
			CronEd.CN_YSel:=CronEd.CN_YSel+Cmd_Buf[8];	//**
//			Cmd_Buf_U16:=ADR(Cmd_Buf[8]); Sostituisco questa riga e la seguente con le 3 precedenti per little/big endian (**)
//			CronEd.CN_YSel:=Cmd_Buf_U16^;
			CronEd.CA_Sel:=Cmd_Buf[10];
			MEMCPY(ADR(Cmd_Buf[11]),ADR(CronEd.CA.Profile),32);
			CronEd.CA_Save_Exe();
		END_IF
		9: (* Active crono immediatly *)
			CronEd.CN_Sel:=WORD_TO_BYTE(Cmd_ObjIdx);
			for x:= 1 to CRON_MAX do
				if CRON[x].ID = CronEd.CN_Sel then
					CRON[x].InitOK:=FALSE;
				end_if
			end_for

ELSE
	Cmd_R:=3;
END_CASE
END_ACTION

ACTION Cmd_GRU:
(* Check index *)(*
IF Cmd_ObjIdx<>1 THEN
	Cmd_R:=2;
	RETURN;
END_IF

(* Process command *)
CASE Cmd_C OF

	1: (* GET CLIMATIC *)
		Cmd_RLen:=20;
		FOR i:=0 TO 4 DO
			j:=DINT_TO_INT(GRU01_Clima.Points[i].X);
			TxLen:=TxLen+RAWTOHEX(ADR(j),2,ADR(TxData[TxLen]));
			j:=DINT_TO_INT(GRU01_Clima.Points[i].Y);
			TxLen:=TxLen+RAWTOHEX(ADR(j),2,ADR(TxData[TxLen]));
		END_FOR

	2: (* SET CLIMATIC *)
		IF Cmd_CLen<>20 THEN
			Cmd_R:=4;
		ELSE
			FOR i:=0 TO 4 DO
				Cmd_Buf_INT:=ADR(Cmd_Buf[8+4*i]); j:=Cmd_Buf_INT^;
				GRU01_Clima.Points[i].X:=INT_TO_DINT(j);
				Cmd_Buf_INT:=ADR(Cmd_Buf[10+4*i]); j:=Cmd_Buf_INT^;
				GRU01_Clima.Points[i].Y:=INT_TO_DINT(j);
			END_FOR
		END_IF

ELSE
	Cmd_R:=3;
END_CASE
*);
END_ACTION

ACTION Cmd_PDC:
(* Check index *)(*
IF Cmd_ObjIdx<>1 THEN
	Cmd_R:=2;
	RETURN;
END_IF

(* Process command *)
CASE Cmd_C OF

	3: (* TRY REARM *)
		PDC01.Rearm:=TRUE;

ELSE
	Cmd_R:=3;
END_CASE
*);
END_ACTION

ACTION Cmd_SYS:
(* Check index *)
IF Cmd_ObjIdx<>0 THEN
	Cmd_R:=2;
	RETURN;
END_IF

(* Process command *)
CASE Cmd_C OF

	0: (* ECHO *)
		IF Cmd_CLen<>0 THEN
			TxLen:=0;
		END_IF

	1: (* LOG REQUEST *)
		LogTrig();

	2: (* REARM *)
		Sys.Warning:=FALSE;
		Sys.Alarm:=FALSE;
		Sys.AlarmStop:=FALSE;

	3: (* GET INFO1 *)
		Cmd_RLen:=6;
		Plant_SN_H:= Plant_SN and 16#FFFF0000;
		Plant_SN_L:= Plant_SN and 16#0000FFFF;
		Plant_SN_H:=shr(Plant_SN_H, 16);
		Plant_SN_H_W:=dword_to_word(Plant_SN_H);
		Plant_SN_H_W:=rol(Plant_SN_H_W, 8);
		Plant_SN_L_W:=dword_to_word(Plant_SN_L);
		Plant_SN_L_W:=rol(Plant_SN_L_W, 8);
		TxLen:=TxLen+RAWTOHEX(ADR(Plant_SN_H_W),2,ADR(TxData[TxLen]));
		TxLen:=TxLen+RAWTOHEX(ADR(Plant_SN_L_W),2,ADR(TxData[TxLen]));
		//TxLen:=TxLen+RAWTOHEX(ADR(Plant_SN),4,ADR(TxData[TxLen]));
		Plant_SW_VER:=rol(Plant_SW_VER, 8);
		TxLen:=TxLen+RAWTOHEX(ADR(Plant_SW_VER),2,ADR(TxData[TxLen]));	
(*
		Cmd_RLen:=6;
		TxLen:=TxLen+RAWTOHEX(ADR(Plant_SN),4,ADR(TxData[TxLen]));
		TxLen:=TxLen+RAWTOHEX(ADR(Plant_SW_VER),2,ADR(TxData[TxLen]));
*)
	14: (* Set data e ora *)
		Year:=byte_to_word(Cmd_Buf[8]); 
		Year:=SHL(Year,8);
		Year:=Year + byte_to_word(Cmd_Buf[9]); 
		Year:=rol(Year, 8);
		Month:=word_to_byte(Cmd_Buf[10]); 
		Day:=word_to_byte(Cmd_Buf[12]); 
		Hour:=word_to_byte(Cmd_Buf[14]); 
		minute:=word_to_byte(Cmd_Buf[16]); 
		Sec:=word_to_byte(Cmd_Buf[18]); 
(*
		Year:=byte_to_word(Cmd_Buf[8]); 
		Year:=SHL(Year,8);
		Year:=Year + byte_to_word(Cmd_Buf[9]); 
		Month:=word_to_byte(Cmd_Buf[11]); 
		Day:=word_to_byte(Cmd_Buf[13]); 
		Hour:=word_to_byte(Cmd_Buf[15]); 
		minute:=word_to_byte(Cmd_Buf[17]); 
		Sec:=word_to_byte(Cmd_Buf[19]); 
*)
		DTStr := concat('DT#',word_to_string(Year));
		DTStr := concat(DTStr,'-');
		DTStr := concat(DTStr,byte_to_string(Month));
		DTStr := concat(DTStr,'-');
		DTStr := concat(DTStr,byte_to_string(Day));
		DTStr := concat(DTStr,'-');
		DTStr := concat(DTStr,byte_to_string(Hour));
		DTStr := concat(DTStr,':');
		DTStr := concat(DTStr,byte_to_string(minute));
		DTStr := concat(DTStr,':');
		DTStr := concat(DTStr,byte_to_string(Sec));
		DateTime:=string_to_dt(DTStr);
		Result:=SysRtcSetTime(DateTime);

ELSE
	Cmd_R:=3;
END_CASE
END_ACTION

ACTION Command:
(* Default response OK/NODATA *)
Cmd_R:=0;
Cmd_RLen:=0;
TxLen:=16;

(* Check object *)
CASE Cmd_Obj OF

	EO_SYS:
		Cmd_SYS();
(*
	EO_GRU:
		Cmd_GRU();

	EO_PDC:
		Cmd_PDC();

	EO_CAL:
		Cmd_CAL();
*)
	EO_CRON:
		Cmd_CRON();

	EO_LUX:
		Cmd_LUX();
		
ELSE
	Cmd_R:=1;
END_CASE

(* Generate response *)
IF TxLen>0 THEN
	Cmd_Obj:=rol(Cmd_Obj, 8); //Scambio byte per compatibilità con sistema wago little endian
	RAWTOHEX(ADR(Cmd_Obj)	,2,ADR(TxData[ 0]));
	Cmd_ObjIdx:=rol(Cmd_ObjIdx, 8); //Scambio byte per compatibilità con sistema wago little endian
	RAWTOHEX(ADR(Cmd_ObjIdx),2,ADR(TxData[ 4]));
	Cmd_R:=rol(Cmd_R, 8); //Scambio byte per compatibilità con sistema wago little endian
	RAWTOHEX(ADR(Cmd_R)		,2,ADR(TxData[ 8]));
	Cmd_RLen:=rol(Cmd_RLen, 8); //Scambio byte per compatibilità con sistema wago little endian
	RAWTOHEX(ADR(Cmd_RLen)	,2,ADR(TxData[12]));
	TxTrig:=TRUE;
END_IF
(*
IF TxLen>0 THEN
	RAWTOHEX(ADR(Cmd_Obj)	,2,ADR(TxData[ 0]));
	RAWTOHEX(ADR(Cmd_ObjIdx),2,ADR(TxData[ 4]));
	RAWTOHEX(ADR(Cmd_R)		,2,ADR(TxData[ 8]));
	RAWTOHEX(ADR(Cmd_RLen)	,2,ADR(TxData[12]));
	TxTrig:=TRUE;
END_IF
*)
END_ACTION

ACTION Cmd_LUX:
(* Check index *)
if Cmd_ObjIdx<1 OR Cmd_ObjIdx>LUXM_MAX then
	Cmd_R:=2; //id del lux fuori range
	return;
end_if

x:=1;
while (Cmd_ObjIdx <> LUXM[x].ID) and ( x <= LUXM_MAX) do
	x := x + 1;	
end_while
if Cmd_ObjIdx = LUXM[x].ID then	
	(* Process command *)
	case Cmd_C of
	
		0:	(* Restore default functioning mode *)
		LUXM[x].TCP_CommandMAN := FALSE; // Spengo il manuale
		if (x<= ACTIVELUX) and (x>0) then 
			LUXM[x].CTRL_MODE:=LUXM[x].CTRL_MODE_backUp;
		end_if
		LUXM[x](WORKINGTIME:=WORKINGTIME[x],POWERONCYCLES:=POWERONCYCLES[x],
													ENERGYCOUNTER:=ENERGYCOUNTER[x], 
													ENERGYCOUNTER_T:=ENERGYCOUNTER_T[x],
													CTRL_EXTON:=KEYON);

		1:	(* Reset statistic counter *)
		LUXM[x].StatReset(WORKINGTIME:=WORKINGTIME[x],POWERONCYCLES:=POWERONCYCLES[x],
															ENERGYCOUNTER:=ENERGYCOUNTER[x], 
															ENERGYCOUNTER_T:=ENERGYCOUNTER_T[x],
															CTRL_EXTON:=KEYON);
	
		2,3:	(* Switch On (command=2) or Off (command=3) lux *)
		case Cmd_C of
			2: (*switch a Manuale ON*)
			LUXM[x].TCP_CommandMAN := TRUE; // Set to Manuale
			LUXM[x].TCP_CommandON := TRUE; // Set to ON
			LUXM[x](WORKINGTIME:=WORKINGTIME[x],POWERONCYCLES:=POWERONCYCLES[x],
														ENERGYCOUNTER:=ENERGYCOUNTER[x], 
														ENERGYCOUNTER_T:=ENERGYCOUNTER_T[x],
														CTRL_EXTON:=KEYON);
			3: (*switch a Manuale OFF*)
			LUXM[x].TCP_CommandMAN := TRUE; // Set to Manuale
			LUXM[x].TCP_CommandON := FALSE; // Set to OFF
			LUXM[x](WORKINGTIME:=WORKINGTIME[x],POWERONCYCLES:=POWERONCYCLES[x],
														ENERGYCOUNTER:=ENERGYCOUNTER[x], 
														ENERGYCOUNTER_T:=ENERGYCOUNTER_T[x],
														CTRL_EXTON:=KEYON);
			
		end_case
		4: (* Modify timer value *)
		if LUXM[x].CTRL_MODE > 0 then //la modifica ha senso per i lux a timer
			NewValueTimerH:=byte_to_word(Cmd_Buf[8]);
			NewValueTimerH:=SHL(NewValueTimerH,8); 
			NewValueTimerH:=NewValueTimerH+byte_to_word(Cmd_Buf[9]);
			NewValueTimerH:=rol(NewValueTimerH, 8);

			NewValueTimerL:=byte_to_word(Cmd_Buf[10]);
			NewValueTimerL:=SHL(NewValueTimerL,8); 
			NewValueTimerL:=NewValueTimerL+byte_to_word(Cmd_Buf[11]);
			NewValueTimerL:=rol(NewValueTimerL, 8);
			
			NewValueTimer:=word_to_dword(NewValueTimerH);			
			NewValueTimer:=SHL(NewValueTimer,16);
			NewValueTimer:=NewValueTimer+word_to_dword(NewValueTimerL);

(*			NewValueTimer:=byte_to_dword(Cmd_Buf[8]);
			NewValueTimer:=SHL(NewValueTimer,8); 
			NewValueTimer:=NewValueTimer+byte_to_dword(Cmd_Buf[9]);
			NewValueTimer:=SHL(NewValueTimer,8); 
			NewValueTimer:=NewValueTimer+byte_to_dword(Cmd_Buf[10]);
			NewValueTimer:=SHL(NewValueTimer,8); 
			NewValueTimer:=NewValueTimer+byte_to_dword(Cmd_Buf[11]);
				//TabLuxPsg[x].TimerOn := dword_to_time(NewValueTimer*1000);
*)
			for x := 1 to LUXM_MAX do
				if LUXM[x].ID = Cmd_ObjIdx
					then LUXM[x].StrLuxTimer := NewValueTimer; //dword_to_time(NewValueTimer*1000); //set del nuovo valore del timer del lux 	
				end_if
			end_for
		else
			Cmd_R:=3; //Comando errato / non previsto
		end_if	 
		5:	(* get working mode*)
			Cmd_RLen:=2;
	//		ModeFromPlc:=LUXM[x].CTRL_MODE; //GIURE gestire con un case ---!!!!!!!!!!!!!!!!!!!!!!!!!!!!
			if LUXM[x].TCP_CommandMAN = TRUE then
				if LUXM[x].TCP_CommandON = TRUE then
					ModeFromPlc:=1;
				elsif LUXM[x].TCP_CommandON = FALSE then
					ModeFromPlc:=0;
				end_if
			elsif  LUXM[x].TCP_CommandMAN = FALSE then
				if ((x<= ACTIVELUX) and (x>0)) then 
					if LUXM[x].CTRL_MODE_backUp > 0 then 
						ModeFromPlc:=3; //timer
					end_if
				else 
					ModeFromPlc:=2; //crono
					//end_if
				end_if
			end_if
			ModeFromPlc:=rol(ModeFromPlc, 8);
			TxLen:=TxLen+RAWTOHEX(ADR(ModeFromPlc),2,ADR(TxData[TxLen]));
			
//		6: (* Modify dimming value for timer control *)
//		7: (* Modify dimming value for key control *)
//		8: (* Modify start and stop orari di funzionamento dei lux a timer *)
	else
		Cmd_R:=3; //Comando errato / non previsto
	end_case
else
	Cmd_R:=2; //id del lux non presente in lista
end_if
END_ACTION

END_PROGRAM

// POUs/TCP_Logger/LogEv
FUNCTION LogEv : BOOL
VAR_INPUT
	Level	: en_Logger_ErrLev;
	Object  : en_SYS_Objects;
	Index	: WORD;
	Error	: WORD;
	Message : STRING;
END_VAR
VAR
	s1 : STRING(160);
	i  : INT;
END_VAR

(* Execute error level operations *)
CASE Level OF
	EL_Wrn: 		Sys.Warning:=TRUE;
	EL_Alarm: 		Sys.Alarm  :=TRUE;
	EL_AlarmStop: 	Sys.Alarm  :=TRUE; (* GO TO STOP STATE!! *)
END_CASE

(* Fill lastlog list *)
s1:=CONCAT(Sys.Time_LogString,';Lev=');
s1:=CONCAT(s1,INT_TO_STRING(Level));
s1:=CONCAT(s1,';Obj=');
s1:=CONCAT(s1,INT_TO_STRING(Object));
s1:=CONCAT(s1,';Idx=');
s1:=CONCAT(s1,WORD_TO_STRING(Index));
s1:=CONCAT(s1,';Err=');
s1:=CONCAT(s1,WORD_TO_STRING(Error));
Sys.LastLogs_Dat[Sys.LastLogs_Idx]:=s1;
Sys.LastLogs_Msg[Sys.LastLogs_Idx]:=Message;
Sys.LastLogs_Idx:=Sys.LastLogs_Idx+1;
IF Sys.LastLogs_Idx>5 THEN Sys.LastLogs_Idx:=0; END_IF

(*---------------------------------------------------------------*)
	Logger_Head();
(*---------------------------------------------------------------*)

(* Insert ERR *)
s1:=CONCAT('&ERR=',INT_TO_STRING(Level));
s1:=CONCAT(s1,';');
s1:=CONCAT(s1,INT_TO_STRING(Object));
s1:=CONCAT(s1,';');
s1:=CONCAT(s1,WORD_TO_STRING(Index));
s1:=CONCAT(s1,';');
s1:=CONCAT(s1,WORD_TO_STRING(Error));
s1:=CONCAT(s1,';');
ADDSTRING(ADR(Logger.TData), ADR(s1), Logger.TLen);
s1:=Message;
STR_NOSPACES(ADR(s1));
ADDSTRING(ADR(Logger.TData), ADR(s1), Logger.TLen);

(*---------------------------------------------------------------*)
	Logger_Send();
(*---------------------------------------------------------------*)

END_FUNCTION

// POUs/TCP_Logger/Logger_Head
FUNCTION Logger_Head : BOOL
VAR
	s1 : STRING(160);
	i  : BYTE;
END_VAR

Logger.TLen:=0;
(* Set GET header *)
ADDSTRING(ADR(Logger.TData), ADR(Logger_GETSTART), Logger.TLen);

(* Insert Header *)
s1:=INSERT('ID=&V=1&D=',DWORD_TO_STRING(Plant_SN),3);
s1:=CONCAT(s1,Sys.Time_LogString);
s1:=CONCAT(s1,'&S=');
IF Sys.Alarm THEN i:=2; ELSIF Sys.Warning THEN i:=1; ELSE i:=0; END_IF
s1:=CONCAT(s1,BYTE_TO_STRING(i));
ADDSTRING(ADR(Logger.TData), ADR(s1), Logger.TLen);

END_FUNCTION

// POUs/Utils Functions/ADDSTRING
FUNCTION ADDSTRING : BOOL (* Append string to a byte buffer *)
VAR_INPUT
	pTxData: POINTER TO BYTE;
	pString: POINTER TO BYTE;
END_VAR
VAR_IN_OUT
	TxLen: DINT;
END_VAR
VAR
END_VAR

pTxData:=pTxData+TxLen;
WHILE pString^<>0 DO
	pTxData^:=pString^;
	pString:=pString+1;
	pTxData:=pTxData+1;
	TxLen:=TxLen+1;
END_WHILE

END_FUNCTION

// POUs/Utils Functions/STR_NOSPACES
FUNCTION STR_NOSPACES : BOOL (* Replace spaces and bad chars with allowed ones, used as HTTP-GET validator *)
VAR_INPUT
	pString: POINTER TO BYTE;
END_VAR
VAR
END_VAR

WHILE pString^<>0 DO
	IF pString^=16#20 (* space *) THEN pString^:=16#5F; (*'_'*) END_IF
	pString:=pString+1;
END_WHILE

END_FUNCTION

// POUs/TCP_Logger/Logger_Send
FUNCTION Logger_Send : BOOL
VAR
	hFile		: RTS_IEC_HANDLE;
	hRes		: RTS_IEC_RESULT;
	pos:	DWORD;
	ts: STRING;
	ts2: STRING;
END_VAR

(* Finalize string *)
ADDSTRING(ADR(Logger.TData), ADR(Logger_GETEND), Logger.TLen);

(* Read log position *)
ts:=Logger_DataFile;
pos:=SysFileGetSize(ts, ADR(hRes));
(* Check log size, bckup and erase if no pending messages *)
IF pos>1000000 THEN
	ts:=Logger_IndexFile;
	hFile:=SysFileOpen(ts,AM_READ,ADR(hRes));
	IF hFile=RTS_INVALID_HANDLE THEN
		ts:=Logger_DataFileOld;
		SysFileDelete(ts);
		ts:=Logger_DataFile; ts2:=Logger_DataFileOld;
		SysFileRename(ts,ts2);
		pos:=0;
	ELSE
		SysFileClose(hFile);
	END_IF
END_IF
(* Write message on log file *)
ts:=Logger_DataFile;
hFile:=SysFileOpen(ts,AM_APPEND_PLUS,ADR(hRes));
IF hFile<>RTS_INVALID_HANDLE THEN
	SysFileWrite(hFile, ADR(Logger.TData), Logger.TLen, ADR(hRes));
	SysFileClose(hFile);
ELSE
	Sys.Warning:=TRUE;
END_IF


(* Check logger status *)
IF Logger.SendReq=FALSE THEN
	(* Set log position for recovery *)
	Logger.SendIdx:=pos;
	(* Copy message data *)
	MEMCPY(ADR(Logger.TData),ADR(Logger.SendData),DINT_TO_WORD(Logger.TLen));
	Logger.SendLen:=Logger.TLen;
	(* Trigger request *)
	Logger.SendReq:=TRUE;
ELSE
	(* Add message position+size in recovery indexes *)
	ts:=Logger_IndexFile;
	hFile:=SysFileOpen(ts, AM_APPEND_PLUS, ADR(hRes));
	SysFileWrite(hFile, ADR(pos), SIZEOF(pos), ADR(hRes));
	SysFileWrite(hFile, ADR(Logger.TLen), SIZEOF(Logger.TLen), ADR(hRes));
	SysFileClose(hFile);
END_IF

END_FUNCTION

// POUs/Utils Functions/MEMCPY
FUNCTION MEMCPY:BOOL
VAR_INPUT
	pSourceAddress:POINTER TO ARRAY[1..2] OF BYTE;
	pDestinationAddress:POINTER TO ARRAY[1..2] OF BYTE;
	BytesToCopy:WORD;
END_VAR
VAR
END_VAR

WHILE (BytesToCopy > 0) DO
	pDestinationAddress^[1]:=pSourceAddress^[1]; (* copy bytes from source to destination *)
	pDestinationAddress:=ADR(pDestinationAddress^[2]); (* increment destination *)
	pSourceAddress:=ADR(pSourceAddress^[2]);(* increment source *)
	BytesToCopy:=BytesToCopy -1; (* decrement number of bytes to copy *)
END_WHILE

END_FUNCTION

// POUs/Utils Functions/HEXTORAW
FUNCTION HEXTORAW : WORD
VAR_INPUT
	pString		: POINTER TO BYTE;
	StringLen	: WORD;
	pData		: POINTER TO BYTE;
END_VAR
VAR
	xl: WORD;
	xi: WORD;
	xr: BYTE;
END_VAR

xl:=0;
xi:=0;

WHILE xi<StringLen DO

	IF pString^>=97 AND pString^<=102 THEN
		xr := pString^ - 87;
	ELSIF pString^>=65 AND pString^<=70 THEN
		xr := pString^ - 55;
	ELSIF pString^>=48 AND pString^<=57 THEN
		xr := pString^ - 48;
	ELSE
		xr := 16;
	END_IF

	IF xr<16 THEN
		IF (xi AND 1)=0 THEN
			pData^ := xr * 16;
		ELSE
			pData^ := pData^ + xr;
			pData := pData + 1;
			xl := xl + 1;
		END_IF
	END_IF

	xi := xi + 1;
	pString := pString + 1;

END_WHILE

HEXTORAW:=xl;

END_FUNCTION

// POUs/Utils Functions/TCPSERVER
FUNCTION_BLOCK TCPSERVER
(***********************************************************************************************************	*)
(* Version: 1.6                                    			          											*)
(* Date: 11.02.2011                                   					          							    *)
(***********************************************************************************************************	*)
(* WAGO Kontakttechnik GmbH Hansastr. 27 32423 Minden(Westf.)													*)
(* Tel. +0049 571/887-0 Fax. +0049 571/887-0																	*)
(* Author: VB																									*)
(***********************************************************************************************************	*)
(*Description:	A TCP server to read and write data													       		*)
(*Historie:																										*)
(*Version 1.6: 11.02.2011: Changes according to 750-880/881											 			*)
(*Version 1.5: 27.11.2008 Bugfix allow reuse port																*)
(*Version 1.4: 13.10.2008 Bugfix transmitting large data														*)
(*Version 1.3: 15.01.2007 Changes according to FW11																*)
(*Version 1.2: 09.03.2006 Changes for socket handle 0											       			*)
(*Version 1.1: 14.02.2005 Release																				*)
(***********************************************************************************************************	*)
VAR CONSTANT
	STATE_INIT     				 : BYTE:= 0;
	STATE_OPEN     				 : BYTE:= 1;
	STATE_TX       				 : BYTE:= 20;
	STATE_RX       				 : BYTE:= 30;
	STATE_CLOSE    				 : BYTE:= 40;
	STATE_ERROR_TRAP		 	 : BYTE:= 200;
END_VAR
VAR_INPUT
	xEnable    					: BOOL;	 (* Set TRUE to enable function block *)
	wPortNumber					: WORD;  (* Port *)
	tServerTimeOut				: TIME:=t#50s;
	ptSendData					: POINTER TO ARRAY[0..MAX_SEND_TCP_SERVER] OF BYTE;
	diSendCount					: DINT;
END_VAR
VAR_OUTPUT
	xClientConnected  			: BOOL:= FALSE;
	diError 					: DINT:= 0;
END_VAR
(* Status Codes -----------------------------------------
	16#8001 => No socket descriptor available 
	16#8002 => SysSockBind fails 
	16#8003 => SysSockListen fails 
	16#8004 => switching to none blocking mode fails
	16#8005 => SysSockClose() returns FALSE 
    16#8006 => SysSockConnect() fails
    16#8007 => SysSockSend() fails
	16#8008 => error state machine 
	16#8009 => timeout while waiting for data from server 
	16#0001 => server waiting for client to establish connection
------------------------------------------------------------*)
VAR_IN_OUT
	xStartSend					: BOOL;
	aReceiveBuffer				: ARRAY [0..MAX_RECEIVE_TCP_SERVER] OF BYTE;
	diReceiveCount				: DINT;
END_VAR

VAR
	m_State    					: BYTE:= 0;
	m_ReceiveBuffer				: ARRAY [0..MAX_RECEIVE_TCP_SERVER_SOCKET] OF BYTE;
	m_ServerSocket				: DINT:= SOCKET_INVALID;
	m_Socket					: DINT:= SOCKET_INVALID;
	m_AddressInfo				: SOCKADDRESS;
	m_BytesReceived				: DINT;
	m_diReturn					: DINT;
	m_xReturn					: BOOL;
	m_SizeSockadr				: DWORD;
	m_ConnectionWatchdog		: TON;
	m_Flags						: DINT;
	m_NoneBlocking   			: DINT:= 1;
	m_Blocking   				: DINT:= 0;
	i							: INT;
	m_count						: DINT;
	diOption					: DINT := 1;
	on: DINT;
END_VAR

IF xEnable THEN
	CASE m_State OF
		STATE_INIT:
			(* Create Socket *)
			m_ServerSocket:= SysSockCreate( SOCKET_AF_INET, SOCKET_STREAM, 0);
			IF m_ServerSocket = SOCKET_INVALID THEN
				(* *)
				diError:= 16#8001;
				m_State:= STATE_ERROR_TRAP;
				RETURN;
			ELSE
				;
			END_IF
			(* Address bindings *)
			(********************)
			on:=1;
			SysSockSetOption( m_ServerSocket, SOCKET_SOL, SOCKET_SO_REUSEADDR, ADR(on), SIZEOF(on) );

			m_AddressInfo.sin_family:= SOCKET_AF_INET;
			m_AddressInfo.sin_port  := SysSockHtons( wPortNumber);
			m_AddressInfo.sin_addr  := SOCKET_INADDR_ANY;
			IF NOT SysSockBind( m_ServerSocket, ADR(m_AddressInfo), SIZEOF(m_AddressInfo)) THEN
				diError:= 16#8002;
				m_State:= STATE_ERROR_TRAP;
				RETURN;
			END_IF
			(* Wait for connections *)
			(************************)
			IF NOT SysSockListen( m_ServerSocket, 1) THEN
				diError:= 16#8003;
				m_State:= STATE_ERROR_TRAP;
			END_IF

			(* Puts SOCKET in NonBlocking mode *)
			m_diReturn:= SysSockIoctl( m_ServerSocket, SOCKET_FIONBIO, ADR(m_NoneBlocking));

			m_State:= STATE_OPEN;


		STATE_OPEN: 	(* Waiting for incomming connection *)
				m_SizeSockadr:=SIZEOF(m_AddressInfo);
				m_Socket:= SysSockAccept( m_ServerSocket, ADR(m_AddressInfo), ADR(m_SizeSockadr));
				diError:=State_open;
				IF m_Socket <> SOCKET_INVALID THEN
					xClientConnected:=TRUE;
					(*Set Push-Bit:new V1.5*)
				(*	IF ADR(%MW0)=16#30000000  OR ADR(%MW0)=16#20000000 THEN (*841 or 881*)
						SysSockSetOption(
							diSocket:=m_Socket,
							diLevel:=6,
							diOption:=SOCKET_TCP_NODELAY,
							pOptionValue:=ADR(diOption),
							diOptionLength:=SIZEOF(diOption));
					ELSE
							;
					END_IF *)
					SysSockIoctl( m_Socket, SOCKET_FIONBIO, ADR(m_NoneBlocking));
					m_State:= STATE_RX;
					diError:=0;
				END_IF

		STATE_RX:
					m_BytesReceived:= SysSockRecv( m_Socket, ADR(m_ReceiveBuffer), SIZEOF(m_ReceiveBuffer), 0);
					CASE m_BytesReceived OF
					-1:(*no data available or error occured*)
						m_ConnectionWatchdog(IN:=TRUE , PT:=T#200ms);	//   T#200ms tServerTimeOut );
						IF m_connectionWatchdog.Q THEN
							m_State:= STATE_CLOSE;
							m_ConnectionWatchdog(IN:=FALSE);(*reset connection watchdog*)
							diError := 16#8009;
						END_IF
					0:(* socket was "gracefully closed"  *)
						m_State:= STATE_CLOSE;
						diError := 16#8003;
					ELSE
						(* Copy received data into receive buffer *)
						(********************************)
						FOR i:= 0 TO DINT_TO_INT(m_BytesReceived	)-1 DO
							aReceiveBuffer[diReceiveCount]:= m_ReceiveBuffer[i];
							diReceiveCount:=(diReceiveCount+1) MOD SIZEOF(aReceiveBuffer);
						END_FOR

						m_ConnectionWatchdog(IN:=FALSE);(*reset connection watchdog*)
					END_CASE

				(*send data*)
				IF xStartSend	 THEN
					m_State := STATE_TX;
				END_IF

	STATE_TX:	 (* send TCP-message *)
		m_diReturn := SysSockSend(diSocket := m_Socket,
								  pbyBuffer := ADR(ptSendData^[m_count]),(*geändert V1.4 bisher: [0] *)
								  diBufferSize := diSendCount-m_count,
								  diFlags :=m_Flags);
		CASE m_diReturn OF
		-1:	(* ERROR or data could not yet be send (V1.3 due to new FW11) *)
			m_ConnectionWatchdog(IN:=TRUE , PT:=tServerTimeOut );
			IF m_connectionWatchdog.Q THEN
				m_State:= STATE_CLOSE;
				m_ConnectionWatchdog(IN:=FALSE);(*reset connection watchdog*)
				diError := 16#8007;
			END_IF
		0: (* socket was "gracefully closed"  *)
			m_State := STATE_CLOSE;
			diError := 16#8003;
		ELSE (* succesful *)
			m_count:=m_count+m_diReturn;
			IF m_count>=diSendCount THEN
				diError := 16#0000;
				m_State := STATE_RX;
				m_count:=0;
				xStartSend:=FALSE;
			END_IF
			m_ConnectionWatchdog(IN:=FALSE);(*reset connection watchdog*)
		END_CASE


		STATE_CLOSE:	(* Close the server *)

	(*		IF ADR(%MW0)=16#30000000  OR ADR(%MW0)=16#20000000 THEN (*841 or 881*)
			;
		ELSE
			IF m_Socket>=0 THEN
				SysSockShutdown(m_Socket, 0);;(*870*)
			END_IF
		END_IF  *)
		IF m_Socket>=0 THEN
			SysSockClose( m_Socket);
		END_IF
		xClientConnected:= FALSE;
		m_State:= STATE_OPEN; (* Try to open the server again *)
		m_ConnectionWatchdog(IN:=FALSE);(*reset connection watchdog*)

		STATE_ERROR_TRAP: (* Error Read/Write socket  *)
			m_State:= STATE_ERROR_TRAP;

	ELSE  (* Bad FSM code trap  *)
			m_State:= STATE_ERROR_TRAP;
			diError:= 16#8008;
	END_CASE;
ELSE
	IF m_State <> STATE_INIT THEN
	(*	IF ADR(%MW0)=16#30000000  OR ADR(%MW0)=16#20000000 THEN (*841 or 881*)
			;
		ELSE
			IF m_Socket>=0 THEN
				SysSockShutdown(m_Socket, 0);;(*870*)
			END_IF
		END_IF *)
		IF m_Socket>=0 THEN
			SysSockClose( m_Socket);
		END_IF
		(*	IF ADR(%MW0)=16#30000000  OR ADR(%MW0)=16#20000000 THEN (*841 or 881*)
			;
		ELSE
			IF m_ServerSocket>=0 THEN
				SysSockShutdown(m_ServerSocket, 0);;(*870*)
			END_IF
		END_IF *)
		IF m_ServerSocket>=0 THEN
			SysSockClose( m_ServerSocket);
		END_IF
		xClientConnected:= FALSE;
		diError:= 0;
		m_State:= STATE_init; (* Try to open the server again *)
		m_ConnectionWatchdog(IN:=FALSE);(*reset connection watchdog*)
	END_IF
END_IF

END_FUNCTION_BLOCK

// POUs/Utils Functions/RAWTOHEX
FUNCTION RAWTOHEX : WORD
VAR_INPUT
	pData: POINTER TO BYTE;
	DataLen: WORD;
	pString: POINTER TO BYTE;
END_VAR
VAR
	xl: WORD;
END_VAR

xl:=0;

WHILE DataLen>0 DO

	pString^ := (pData^ / 16#10) + 48 + (((pData^ / 16#10)/10)*7);
	pString:=pString+1;
	pString^ := (pData^ AND 16#0F)  + 48 + (((pData^ AND 16#0F)/10)*7);
	pString:=pString+1;
	pData:=pData+1;
	DataLen:=DataLen-1;
	xl:=xl+2;

END_WHILE

(*pString^:=0;*)

RAWTOHEX:=xl;

END_FUNCTION

// POUs/TCP_Logger/LogTrig
FUNCTION LogTrig : BOOL
VAR
	s1 : STRING(160);
	i  : BYTE;
END_VAR

(*---------------------------------------------------------------*)
	Logger_Head();
(*---------------------------------------------------------------*)

(* Log PSG values *)
(* 
s1:=CONCAT('&PSG=',DWORD_TO_STRING(PASSAGES[1]));
FOR i := 2 TO PSG_MAX DO
	s1:=CONCAT(s1,';');
	s1:=CONCAT(s1,DWORD_TO_STRING(PASSAGES[i]));
END_FOR
ADDSTRING(ADR(Logger.TData), ADR(s1), Logger.TLen);
 *)
for i := 1 TO PSG_MAX DO	
	if PSG[i].ID <> 0
	then PSG[i].AddLogData(PASSAGES:=PASSAGES[i]);	//PSG[i].AddLogData(NumTransition:=PsgCounter[PSG[i].ID]);
 	end_if
END_FOR


(* Log LUXM *)
FOR i := 1 TO LUXM_MAX DO
	LUXM[i].AddLogData(WORKINGTIME:=WORKINGTIME[i], POWERONCYCLES:=POWERONCYCLES[i],
					   ENERGYCOUNTER:=ENERGYCOUNTER[i], ENERGYCOUNTER_T:=ENERGYCOUNTER_T[i]);
END_FOR

(* Log ZREL *)
FOR i := 1 TO ZREL_MAX DO
	ZREL[i].AddLogData(MODBUS:=MODB01);
END_FOR

(* Log CRON *)
//GIURE ver 21 - Eseguo log crono dal 18 al 38 (da 1 a 17 non sono soggette a crono)
FOR i := 1 TO CRON_MAX DO
	if CRON[i].ID <> 0
		then CRON[i].AddLogData(SET_POINT:=CRON[i].SetPoint, STAT_LOG:=CRON[i].Status_Log);
	end_if
END_FOR

(*---------------------------------------------------------------*)
	Logger_Send();
(*---------------------------------------------------------------*)

END_FUNCTION

// POUs/TCP_Logger/Logger_Proc
PROGRAM Logger_Proc
VAR
	c1:         	TCPCLIENT;

	Open:	    	BOOL;
	IpAddr:			DWORD;
	InetAddr:		DWORD;
	Connected:  	BOOL;
	Error:      	DINT;
	TxTrig:     	BOOL;
	RxData:			ARRAY [0..MAX_RECEIVE_TCP_CLIENT] OF BYTE;
	RxLen:			DINT;

	Retry:			BYTE;	(* Counter for connection retries *)
	Recovered:		BYTE;	(* Counter for recovered unsent messages *)

	i:				DINT;
	pos:			DWORD;
	hFile		: RTS_IEC_HANDLE;
	hRes		: RTS_IEC_RESULT;
	ts: STRING;
END_VAR

(*=== State machine ===*)
CASE Logger.Status OF

	S_Logger_UNKNOWN:
		(* Startup *)
		Logger.SendReq:=FALSE;
		Open:=FALSE;
		Logger.Status:=S_Logger_IDLE;

	S_Logger_IDLE:
		(* Wait request *)
		IF Logger.SendReq THEN
			(* Resolve server name or use static IP *)
			IF LEN(Logger_SERVER)=0 THEN
				ts:=Logger_IP;
				InetAddr:=SysSockInetAddr(ts);
			ELSE
				ts:=Logger_SERVER;
				IpAddr:=SysSockGetHostByName(ts);
				DWORDSWAP(pIn:=ADR(IpAddr), pOut:=ADR(InetAddr));
			END_IF
			TxTrig:=FALSE;
			RxLen:=0;
			(* Open connection *)
			Open:=TRUE;
			Logger.Status:=S_Logger_WAITCONN;
		END_IF

	S_Logger_WAITCONN:
		(* Wait connection *)
		IF Connected THEN
			(* Send data *)
			TxTrig:=TRUE;
			Logger.Status:=S_Logger_WAITTX;
		END_IF
		IF Error>0 THEN
			Open:=FALSE;
			Logger.Status:=S_Logger_ERROR;
		END_IF

	S_Logger_WAITTX:
		(* Wait transmission *)
		IF NOT TxTrig THEN
			Logger.Status:=S_Logger_WAITRESP;
		END_IF
		IF Error>0 THEN
			Open:=FALSE;
			Logger.Status:=S_Logger_ERROR;
		END_IF

	S_Logger_WAITRESP:
		(* Wait response *)
		IF Connected=FALSE OR RxLen>=4 THEN
			Open:=FALSE;
			(* Check response *)
			IF RxLen>=4 AND CHKSTRING(pString:=ADR(RxData), pPattern:=ADR(Logger_CHECK)) THEN
				Logger.SendReq:=FALSE;
				Retry:=0;
				(* Check unsent messages to flush *)
				IF Recovered<Logger_RecoverMsgs THEN
					MsgChk();
					IF Logger.SendReq=TRUE THEN
						Recovered:=Recovered+1;
					ELSE
						Recovered:=0;
					END_IF
				ELSE
					Recovered:=0;
				END_IF
				Logger.Status:=S_Logger_IDLE;
			ELSE
				Logger.Status:=S_Logger_ERROR;
			END_IF
		END_IF

	S_Logger_ERROR:
		(* Connection error or send failure *)
		Retry:=Retry+1;
		IF Retry>Logger_ConnRetries THEN
			(* Save message as unsent *)
			MsgSave();
			Logger.SendReq:=FALSE;
			Retry:=0;
		END_IF
		Logger.Status:=S_Logger_IDLE;

ELSE
	Logger.Status:=S_Logger_UNKNOWN;
END_CASE


(*=== Execute client lib ===*)
c1(
	xOpenConnection			:= Open,
	dwInetAddr 				:= InetAddr,
	wPortNumber				:= Logger_PORT,
	ptSendData				:= ADR(Logger.SendData),
	diSendCount				:= Logger.SendLen,
	tConnectWatchdogTime	:= T#20S, //t#10s,
	xStartSend				:= TxTrig,
	aReceiveBuffer			:= RxData,
	diReceiveCount			:= RxLen,
	xConnected				=> Connected,
	diError					=> Error
);

(*=== Process Rx data ===*)
(*IF RxLen>0 THEN
	RxLen:=0;
END_IF*)

ACTION MsgChk:
(* Open index file *)
ts:=Logger_IndexFile;
hFile:=SysFileOpen(ts,AM_READ,ADR(hRes));
IF hFile=RTS_INVALID_HANDLE THEN
	RETURN;
END_IF
(* Search oldest message to recover *)
SysFileSetPos(hFile,Logger.LastIdxPos);
Logger.SendLen:=0;
REPEAT
	SysFileRead(hFile, ADR(Logger.SendIdx), SIZEOF(Logger.SendIdx), ADR(hRes));
	SysFileGetPos(hFile, ADR(pos));
	SysFileRead(hFile, ADR(Logger.SendLen), SIZEOF(Logger.SendLen), ADR(hRes));
	hRes:=SysFileEOF(hFile);
UNTIL
	hRes=16#0 OR Logger.SendLen<>0
END_REPEAT
SysFileClose(hFile);
(* Delete index file when all messages are recovered *)
IF Logger.SendLen=0 THEN
	Logger.LastIdxPos:=0;
	ts:=Logger_IndexFile;
	SysFileDelete(ts);
	RETURN;
END_IF
(* Recover message data *)
ts:=Logger_DataFile;
hFile:=SysFileOpen(ts,AM_READ,ADR(hRes));
IF hFile<>RTS_INVALID_HANDLE THEN
	SysFileSetPos(hFile,Logger.SendIdx);
	SysFileRead(hFile,ADR(Logger.SendData),Logger.SendLen,ADR(hRes));
	Logger.SendReq:=TRUE;
	SysFileClose(hFile);
END_IF
(* Clear index entry *)
ts:=Logger_IndexFile;
hFile:=SysFileOpen(ts,AM_READ_PLUS,ADR(hRes));
IF hFile<>RTS_INVALID_HANDLE THEN
	SysFileSetPos(hFile,pos);
	i:=0;
	SysFileWrite(hFile, ADR(i), 4, ADR(hRes));
	SysFileGetPos(hFile,ADR(Logger.LastIdxPos));
	SysFileClose(hFile);
END_IF
END_ACTION

ACTION MsgSave:
(* Add log position in recovery indexes *)
ts:=Logger_IndexFile;
hFile:=SysFileOpen(ts, AM_APPEND_PLUS, ADR(hRes));
SysFileWrite(hFile, ADR(Logger.SendIdx), SIZEOF(Logger.SendIdx), ADR(hRes));
SysFileWrite(hFile, ADR(Logger.SendLen), SIZEOF(Logger.SendLen), ADR(hRes));
SysFileClose(hFile);
END_ACTION

END_PROGRAM

// POUs/Utils Functions/DWORDSWAP
FUNCTION DWORDSWAP:BOOL
VAR_INPUT
	pIn:POINTER TO ARRAY[1..4] OF BYTE;
	pOut:POINTER TO ARRAY[1..4] OF BYTE;
END_VAR
VAR
END_VAR

pOut^[1]:=pIn^[4];
pOut^[2]:=pIn^[3];
pOut^[3]:=pIn^[2];
pOut^[4]:=pIn^[1];

END_FUNCTION

// POUs/Utils Functions/CHKSTRING
FUNCTION CHKSTRING : BOOL
VAR_INPUT
	pString: POINTER TO BYTE;
	pPattern: POINTER TO BYTE;
END_VAR
VAR
END_VAR

CHKSTRING:=TRUE;
WHILE pPattern^<>0 AND CHKSTRING DO
	IF pPattern^<>pString^ THEN CHKSTRING:=FALSE; END_IF
	pString:=pString+1;
	pPattern:=pPattern+1;
END_WHILE

END_FUNCTION

// POUs/Utils Functions/TCPCLIENT
FUNCTION_BLOCK TCPCLIENT
(***********************************************************************************************************	*)
(* Version: 1.3b                        			          													*)
(* Date: 28.10.2014                   				          							            			*)
(***********************************************************************************************************	*)
(* WAGO Kontakttechnik GmbH Hansastr. 27 32423 Minden(Westf.)													*)
(* Tel. +0049 571/887-0 Fax. +0049 571/887-0																	*)
(* Author: VB																									*)
(***********************************************************************************************************	*)
(*Description:	A TCP client to read and write data with additional connection watchdog							*)
(*History:																										*)
(*Version 1.3b: 28.10.2014: Use DWORD address for IP (Andrea Ravasio)											*)
(*Version 1.3: 11.02.2011: Changes according to 750-880/881											 			*)
(*Version 1.2: 29.08.2007 Bugfix TCP Client																		*)
(*Version 1.1: 15.01.2007 Changes according to FW11																*)
(*Version 1.0: 09.03.2006 Release																				*)
(***********************************************************************************************************	*)
VAR CONSTANT
	STATE_CREATE     				 : BYTE:= 0;
	STATE_OPEN     					 : BYTE:= 1;
	STATE_IOCTL    					 : BYTE:= 2;
	STATE_CONNECT     				 : BYTE:= 10;
	STATE_TX       					 : BYTE:= 20;
	STATE_RX       					 : BYTE:= 30;
	STATE_CLOSE    					 : BYTE:= 40;
	STATE_ERROR_TRAP			     : BYTE:= 200;
END_VAR

VAR_INPUT
	xOpenConnection					: BOOL;
	dwInetAddr						: DWORD; (* <== Use SysSockInetAddr() value or
													swapped bytes order of SysSockGetHostByName() value *)
	wPortNumber						: WORD;
	ptSendData						: POINTER TO ARRAY[0..MAX_SEND_TCP_CLIENT] OF BYTE;
	diSendCount						: DINT;
	tConnectWatchdogTime		    : TIME := t#10s;
END_VAR
VAR_OUTPUT
	xConnected						: BOOL;
	diError 						: DINT := 0;
END_VAR
(* ErrorCodes -----------------------------------------
	16#8001 => No socket descriptor available 
	16#8002 => SysSockSend returns -1 
	16#8003 => Socket was "gracefully closed" 
	16#8004 => switching to none blocking mode fails
	16#8005 => SysSockClose() returns FALSE 
    16#8006 => SysSockConnect() fails
    16#8007 => SysSockSend() fails
	16#8008 => error state machine 
	16#8009 => timeout while waiting for data from server 
------------------------------------------------------------*)
VAR_IN_OUT
	xStartSend							: BOOL;
	aReceiveBuffer						: ARRAY [0..MAX_RECEIVE_TCP_CLIENT] OF BYTE;
	diReceiveCount						: DINT;
END_VAR
VAR
	m_State								: BYTE := 0;
	m_ReceiveBuffer						: ARRAY [0..MAX_RECEIVE_TCP_CLIENT_SOCKET] OF BYTE;
	m_Socket							: DINT;
	m_AddressInfo						: SOCKADDRESS;
	m_BytesReceived						: DINT;
	m_diReturn							: DINT;
	m_xReturn							: BOOL;
	m_IoCtlParameter  					: DINT := 1; (* IOCTL-Parameter for non-blocking mode of sockets *)
	i									: INT;
	T_Connect							: TON;
	m_count								: DINT;
	diOption							: DINT := 1;
	m_Blocking   						: DINT := 0;
END_VAR

IF xOpenConnection THEN
	(* State maschine *)
	CASE  m_State OF

	(* -------------------------------------------------------------------------*)
	STATE_CREATE:
			(* create socket descriptor*)
			m_Socket := SysSockCreate(diAddressFamily	:= SOCKET_AF_INET,
													 diType		:= SOCKET_STREAM,
													 diProtocol := SOCKET_IPPROTO_TCP);
			IF m_Socket >= 0 THEN
			(*Set Push-Bit*)
				IF ADR(%MW0)=16#30000000  OR ADR(%MW0)=16#20000000 THEN (*841 or 881*)
					SysSockSetOption(
						diSocket:=m_Socket,
						diLevel:=6,
						diOption:=SOCKET_TCP_NODELAY,
						pOptionValue:=ADR(diOption),
						diOptionLength:=SIZEOF(diOption));
				ELSE
						;
				END_IF
				m_State := STATE_IOCTL; (* succesful *)
			ELSE
				diError := 16#8001;  (* no socket descriptor available *)
				m_State := STATE_ERROR_TRAP;
			END_IF

	(* -------------------------------------------------------------------------*)
	STATE_IOCTL: (* change  socket mode  to none blocking *)
		m_diReturn := SysSockIoctl( m_Socket, SOCKET_FIONBIO, ADR(m_IoCtlParameter));
		//IF m_diReturn <> 0 THEN
			m_AddressInfo.sin_family := SOCKET_AF_INET;
			m_AddressInfo.sin_port := SysSockNtohs(wPortNumber);
			m_AddressInfo.sin_addr := dwInetAddr;
			m_State := STATE_CONNECT;
		//ELSE
		//	diError := 16#8004;  (* switching to none blocking mode fails *)
		//	m_State := STATE_ERROR_TRAP;
		//END_IF


	(* -------------------------------------------------------------------------*)
	STATE_CONNECT: (* connect with server *)
		T_Connect(IN:=TRUE , PT:=tConnectWatchdogTime);(*activate watchdog for establishing connection to a server*)
		m_xReturn := SysSockConnect ( m_Socket, ADR(m_AddressInfo),  SIZEOF(m_AddressInfo));
		IF m_xReturn THEN (* succesful *)
			IF xStartSend THEN
				m_State := STATE_TX;(*transmit data*)
			ELSE
				m_State := STATE_RX;(*wait for data from server*)
			END_IF
			xConnected:=TRUE;
			T_Connect(IN:=FALSE);
		ELSE
			IF T_Connect.Q THEN
				diError := 16#8006;  (* connect fails *)
				xConnected:=FALSE;
				T_Connect(IN:=FALSE);
				m_State := STATE_ERROR_TRAP;
				SysSockClose( m_Socket);
			ELSE
				m_State := STATE_CONNECT;(*client still  tries to set up connection*)
			END_IF
		END_IF


	STATE_TX:	 (* send TCP-message *)
		m_diReturn := SysSockSend(diSocket := m_Socket,
								  pbyBuffer := ADR(ptSendData^[0]),
								  diBufferSize := diSendCount-m_count,
								  diFlags := 0);

		CASE m_diReturn OF
		-1:	(* ERROR *)
			T_Connect(IN:=TRUE , PT:=CONNECT_WATCHDOG_TIME);(*activate watchdog to check communication*)
			IF t_Connect.Q THEN
				diError := 16#8007;
				T_Connect(IN:=FALSE);
				m_State:=STATE_CLOSE;
			END_IF
		0: (* socket was "gracefully closed" *)
			m_State := STATE_CLOSE;
			diError := 16#8003;
		ELSE (* succesful *)
			m_count:=m_count+m_diReturn;
			IF m_count>=diSendCount THEN
				diError := 16#0000;
				m_State := STATE_RX;
				m_count:=0;
				xStartSend:=FALSE;
			END_IF
			T_Connect(IN:=FALSE);
		END_CASE

	(* -------------------------------------------------------------------------*)
	STATE_RX: (* process receive data *)
			m_BytesReceived := SysSockRecv(	diSocket 	:= m_Socket,
										pbyBuffer 	:= ADR(m_ReceiveBuffer),		(* Address of receive buffer *)
										diBufferSize:= SIZEOF(m_ReceiveBuffer),
										diFlags		:= 0);

			CASE m_BytesReceived OF
			-1:	(* No data available or error occured *)
				T_Connect(IN:=TRUE , PT:=tConnectWatchdogTime);(*activate watchdog to check communication*)
				IF t_Connect.Q THEN
					diError:=16#8009;
					T_Connect(IN:=FALSE);
					m_State:=STATE_CLOSE;
				END_IF
				IF xStartSend THEN
					m_State:=STATE_TX	;(* WAIT IN THIS STATE  and check for arriving data or new send command*)
				END_IF;
			0: (* socket was "gracefully closed"  *)
				m_State:=STATE_CLOSE;
				diError := 16#8003;
			ELSE (* succesful *)
				diError := 16#0000;
				T_Connect(IN:=FALSE);
				(* Copy received data into receive buffer *)
				FOR i:= 0 TO DINT_TO_INT(m_BytesReceived	)-1 DO
					aReceiveBuffer[diReceiveCount]:= m_ReceiveBuffer[i];
					diReceiveCount:=(diReceiveCount+1) MOD SIZEOF(aReceiveBuffer);
				END_FOR

			END_CASE

	(* -------------------------------------------------------------------------*)
	STATE_CLOSE : (* close socket *)
		IF ADR(%MW0)=16#30000000  OR ADR(%MW0)=16#20000000 THEN (*841 or 881*)
			;
		ELSE
			SysSockShutdown(m_Socket, 0);;(*870*)
		END_IF
		m_xReturn := SysSockClose( m_Socket);
		m_Socket := -1;
		m_State := 0; (* succesful *)
		xConnected:=FALSE;
		T_Connect(IN:=FALSE);
	(* -------------------------------------------------------------------------*)
	STATE_ERROR_TRAP: (* error handling *)
		xConnected:=FALSE;

	ELSE  (* Bad FSM code trap  *)
			m_State:= STATE_ERROR_TRAP;
			diError:= 16#8008;
	END_CASE

ELSE(*close connection*)
	IF m_Socket >= 0 THEN
		IF ADR(%MW0)=16#30000000  OR ADR(%MW0)=16#20000000 THEN (*841 or 881*)
			;
		ELSE
			SysSockShutdown(m_Socket, 0);;(*870*)
		END_IF
		SysSockClose( m_Socket);
	END_IF
	m_Socket := -1;
	diError := 16#0000;
	m_State := STATE_CREATE;
	xConnected:=FALSE;
	T_Connect(IN:=FALSE);
END_IF

END_FUNCTION_BLOCK

// POUs/Utils/RTC_Update
FUNCTION RTC_Update : BOOL
VAR
	T: DT;
	TS: STRING;
	TS2: STRING;
	Hour: BYTE;
	Minute: BYTE;
END_VAR

(* Get RTC time *)
T:=SysRtcGetTime(TRUE);
Sys.Time_CT_DT:=T;
(* Calculate variables *)
TS:=DT_TO_STRING(T);
Sys.Time_LogString:=DELETE(STR:=TS, LEN:=3, POS:=1);
TS2:=MID(STR:=TS, LEN:=4, POS:= 4); Sys.Time_Year 	:=STRING_TO_WORD(TS2);
TS2:=MID(STR:=TS, LEN:=2, POS:= 9); Sys.Time_Month	:=STRING_TO_BYTE(TS2);
TS2:=MID(STR:=TS, LEN:=2, POS:=12); Sys.Time_Day  	:=STRING_TO_BYTE(TS2);
Sys.Time_CT_Day:=(32*(Sys.Time_Month-1)+Sys.Time_Day-1);
TS2:=MID(STR:=TS, LEN:=2, POS:=15); Hour			:=STRING_TO_BYTE(TS2);
TS2:=MID(STR:=TS, LEN:=2, POS:=18); Minute		 	:=STRING_TO_BYTE(TS2);
Sys.Time_CT_Quarter:=Hour*4+(Minute/15);

END_FUNCTION

// POUs/Utils/CSV_Log
FUNCTION CSV_Log : BOOL
VAR_INPUT
END_VAR
VAR CONSTANT
	LogFileName:STRING:='S:\LOGS_ID4V3.CSV';
END_VAR
VAR
	s1 : STRING(256);
	hFile: 	DWORD;
END_VAR

(* Check file presence *)
hFile:=SysFileOpen(LogFileName,'r');
IF hFile=0 THEN
	(*** File not exist *** Create file and write header *)
	hFile:=SysFileOpen(LogFileName,'w');
	IF hFile<>0 THEN
		(* Write CSV header *)
		s1:='Title1;Title2,...';
		SysFileWrite(hFile, ADR(s1), LEN(s1));
		SysFileWrite(hFile, ADR(Logger_CRLF), LEN(Logger_CRLF));
	END_IF
ELSE
	(*** File exist *** Close file and reopen in append mode *)
	SysFileClose(hFile);
	hFile:=SysFileOpen(LogFileName,'a');
END_IF

(* Log to file *)
IF hFile<>0 THEN
	(* Date stamp *)
	s1:=REPLACE( Sys.Time_LogString , ' ' , 1 , 11 );
	SysFileWrite(hFile, ADR(s1), LEN(s1));
	(* Write CSV data *)
	s1:=CONCAT(';', 'Data1' );
	s1:=CONCAT(s1 , ';');
	s1:=CONCAT(s1 , 'Data2' );
	s1:=CONCAT(s1 , ';');
	s1:=CONCAT(s1 , '...' );
	SysFileWrite(hFile, ADR(s1), LEN(s1));
	(* Add line CRLF and close *)
	SysFileWrite(hFile, ADR(Logger_CRLF), LEN(Logger_CRLF));
	SysFileClose(hFile);
END_IF

END_FUNCTION

// POUs/PLC_RT
PROGRAM PLC_RT
VAR
END_VAR

(******************************************************************************
 ****                       HP TASK CODE	                               ****
 ******************************************************************************
*)

(*==============================*)
(*== Running cycle operations ==*)
(*==============================*)
IF SYS.Status>S_INIT_VAR THEN
	(* Execute cycle processes *)
	PSG[ 1](PSG_IN:=PSG01_IN, PASSAGES:=PASSAGES[ 1]);
	PSG[ 2](PSG_IN:=PSG02_IN, PASSAGES:=PASSAGES[ 2]);
	PSG[ 3](PSG_IN:=PSG03_IN, PASSAGES:=PASSAGES[ 3]);
	PSG[ 4](PSG_IN:=PSG04_IN, PASSAGES:=PASSAGES[ 4]);
	PSG[ 5](PSG_IN:=PSG05_IN, PASSAGES:=PASSAGES[ 5]);
	PSG[ 6](PSG_IN:=PSG06_IN, PASSAGES:=PASSAGES[ 6]);
	PSG[ 7](PSG_IN:=PSG07_IN, PASSAGES:=PASSAGES[ 7]);
	PSG[ 8](PSG_IN:=PSG08_IN, PASSAGES:=PASSAGES[ 8]);
	PSG[ 9](PSG_IN:=PSG09_IN, PASSAGES:=PASSAGES[ 9]);
	PSG[10](PSG_IN:=PSG10_IN, PASSAGES:=PASSAGES[10]);
	PSG[11](PSG_IN:=PSG11_IN, PASSAGES:=PASSAGES[11]);
	PSG[12](PSG_IN:=PSG12_IN, PASSAGES:=PASSAGES[12]);
	PSG[13](PSG_IN:=PSG13_IN, PASSAGES:=PASSAGES[13]);
	PSG[14](PSG_IN:=PSG14_IN, PASSAGES:=PASSAGES[14]);
	PSG[15](PSG_IN:=PSG15_IN, PASSAGES:=PASSAGES[15]);
	PSG[16](PSG_IN:=PSG16_IN, PASSAGES:=PASSAGES[16]);
	PSG[17](PSG_IN:=PSG17_IN, PASSAGES:=PASSAGES[17]);
	PSG[18](PSG_IN:=PSG18_IN, PASSAGES:=PASSAGES[18]);
	PSG[19](PSG_IN:=PSG19_IN, PASSAGES:=PASSAGES[19]);
	PSG[20](PSG_IN:=PSG20_IN, PASSAGES:=PASSAGES[20]);
	PSG[21](PSG_IN:=PSG21_IN, PASSAGES:=PASSAGES[21]);
	PSG[22](PSG_IN:=PSG22_IN, PASSAGES:=PASSAGES[22]);
	PSG[23](PSG_IN:=PSG23_IN, PASSAGES:=PASSAGES[23]);
	PSG[24](PSG_IN:=PSG24_IN, PASSAGES:=PASSAGES[24]);
	PSG[25](PSG_IN:=PSG25_IN, PASSAGES:=PASSAGES[25]);
	PSG[26](PSG_IN:=PSG26_IN, PASSAGES:=PASSAGES[26]);
	PSG[27](PSG_IN:=PSG27_IN, PASSAGES:=PASSAGES[27]);
	PSG[28](PSG_IN:=PSG28_IN, PASSAGES:=PASSAGES[28]);
	PSG[29](PSG_IN:=PSG29_IN, PASSAGES:=PASSAGES[29]);
	PSG[30](PSG_IN:=PSG30_IN, PASSAGES:=PASSAGES[30]);
	PSG[31](PSG_IN:=PSG31_IN, PASSAGES:=PASSAGES[31]);
	PSG[32](PSG_IN:=PSG32_IN, PASSAGES:=PASSAGES[32]);
	PSG[33](PSG_IN:=PSG33_IN, PASSAGES:=PASSAGES[33]);
	PSG[34](PSG_IN:=PSG34_IN, PASSAGES:=PASSAGES[34]);
END_IF

END_PROGRAM

// POUs/Utils Functions/AVERAGE_DINT
FUNCTION_BLOCK AVERAGE_DINT
VAR_INPUT
	IN: 	DINT;
END_VAR
VAR_OUTPUT
	HI:		DINT;
	AVG:	DINT;
	LOW:	DINT;
	ERR:	BOOL;
END_VAR
VAR
	sum:	REAL;
	cnt:	WORD;
END_VAR

IF cnt>=65000 THEN
	ERR:=TRUE;
	Read();
	sum := sum - DINT_TO_REAL(AVG);
	cnt := cnt - 1;
END_IF

sum := sum + DINT_TO_REAL(IN);
cnt := cnt + 1;

IF IN<LOW THEN LOW:=IN; END_IF
IF IN>HI  THEN HI :=IN; END_IF

ACTION Read:
AVG := REAL_TO_DINT(sum/cnt);
END_ACTION

ACTION Reset:
HI:=IN;
AVG:=IN;
LOW:=IN;
ERR:=FALSE;

sum:=DINT_TO_REAL(IN);
cnt:=1;
END_ACTION

END_FUNCTION_BLOCK

// POUs/Utils Functions/AVERAGE_INT
FUNCTION_BLOCK AVERAGE_INT
VAR_INPUT
	IN: 	INT;
END_VAR
VAR_OUTPUT
	HI:		INT;
	AVG:	INT;
	LOW:	INT;
	ERR:	BOOL;
END_VAR
VAR
	sum:	DINT;
	cnt:	WORD;
END_VAR

IF cnt>=65000 THEN
	ERR:=TRUE;
	Read();
	sum := sum - AVG;
	cnt := cnt - 1;
END_IF

sum := sum + IN;
cnt := cnt + 1;

IF IN<LOW THEN LOW:=IN; END_IF
IF IN>HI  THEN HI :=IN; END_IF

ACTION Read:
AVG := DINT_TO_INT(sum/cnt);
END_ACTION

ACTION Reset:
HI:=IN;
AVG:=IN;
LOW:=IN;
ERR:=FALSE;

sum:=IN;
cnt:=1;
END_ACTION

END_FUNCTION_BLOCK

// POUs/Utils Functions/AVERAGE_T
FUNCTION_BLOCK AVERAGE_T
VAR_INPUT
	IN: 	INT;
END_VAR
VAR_OUTPUT
	HI:		INT;
	AVG:	INT;
	LOW:	INT;
	ERR:	BOOL;
END_VAR
VAR
	sum:	DINT;
	cnt:	WORD;
END_VAR

IF cnt>=65000 THEN
	ERR:=TRUE;
	Read();
	sum := sum - AVG;
	cnt := cnt + 1;
END_IF

sum := sum + IN;
cnt := cnt + 1;

IF IN<LOW THEN  LOW:=IN; END_IF
IF IN>HI  THEN HI :=IN; END_IF

ACTION Read:
AVG := DINT_TO_INT(sum/cnt);
END_ACTION

ACTION Reset:
HI:=IN;
AVG:=IN;
LOW:=IN;
ERR:=FALSE;

sum:=IN;
cnt:=1;
END_ACTION

END_FUNCTION_BLOCK

// POUs/Utils Functions/COPY_32SWAP16
FUNCTION COPY_32SWAP16:BOOL
VAR_INPUT
	pSourceAddress		:POINTER TO ARRAY[1..2] OF WORD;
	pDestinationAddress	:POINTER TO ARRAY[1..2] OF WORD;
END_VAR
VAR
END_VAR

pDestinationAddress^[1]:=pSourceAddress^[2];
pDestinationAddress^[2]:=pSourceAddress^[1];

END_FUNCTION

// POUs/Utils Functions/FLT_EVENT
FUNCTION_BLOCK FLT_EVENT
VAR_INPUT
	IN		: BOOL;
	INITEV	: BOOL:=TRUE;
END_VAR
VAR_OUTPUT
	EVH		: BOOL;
	EVL		: BOOL;
END_VAR
VAR
	init	: BOOL:=FALSE;
	old		: BOOL;
END_VAR

EVH:=FALSE;
EVL:=FALSE;

IF NOT init THEN
	init:=TRUE;
	IF INITEV THEN
		old := NOT IN;
	ELSE
		old := IN;
	END_IF
END_IF

IF old<>IN THEN
	old:=IN;
	IF IN THEN EVH:=TRUE; ELSE EVL:=TRUE; END_IF
END_IF

END_FUNCTION_BLOCK

// POUs/Utils Functions/FLT_TAP
FUNCTION_BLOCK FLT_TAP
VAR_INPUT
	IN		: BOOL;
	TAP		: BYTE:=4;
	INITEV	: BOOL:=TRUE;
END_VAR
VAR_OUTPUT
	OUT		: BOOL;
	EVH		: BOOL;
	EVL		: BOOL;
END_VAR
VAR
	init	: BOOL:=FALSE;
	cnt		: BYTE;
END_VAR

EVH:=FALSE;
EVL:=FALSE;

IF NOT init THEN
	init := TRUE;
	IF INITEV THEN
		OUT  := NOT IN;
		cnt  := TAP;
	ELSE
		OUT  := IN;
	END_IF
END_IF

IF OUT<>IN THEN
	cnt:=cnt+1;
	IF cnt>TAP THEN
		OUT:=IN;
		cnt:=0;
		IF OUT THEN EVH:=TRUE; ELSE EVL:=TRUE; END_IF
	END_IF
ELSE
	cnt:=0;
END_IF

END_FUNCTION_BLOCK

// POUs/Utils Functions/FLT_TIME
FUNCTION_BLOCK FLT_TIME
VAR_INPUT
	IN		: BOOL;
	TTAP	: TIME:=T#5s;
	INITEV	: BOOL:=TRUE;
END_VAR
VAR_OUTPUT
	OUT		: BOOL;
	EVH		: BOOL;
	EVL		: BOOL;
END_VAR
VAR
	init	: BOOL:=FALSE;
	timer	: TON;
END_VAR

EVH:=FALSE;
EVL:=FALSE;

IF NOT init THEN
	init := TRUE;
	IF INITEV THEN
		OUT  := NOT IN;
	ELSE
		OUT  := IN;
	END_IF
END_IF

IF OUT<>IN THEN
	timer(IN:=TRUE,PT:=TTAP);
	IF timer.Q THEN
		OUT:=IN;
		timer(IN:=FALSE);
		IF OUT THEN EVH:=TRUE; ELSE EVL:=TRUE; END_IF
	END_IF
ELSE
	timer(IN:=FALSE);
END_IF

END_FUNCTION_BLOCK

// POUs/Utils Functions/LINEAR
FUNCTION LINEAR : REAL (* Linear interpolation *)
VAR_INPUT
	X_In	: REAL;
	P1_X	: REAL;
	P1_Y	: REAL;
	P2_X	: REAL;
	P2_Y	: REAL;
END_VAR
VAR
END_VAR

LINEAR:=P1_Y+(((P2_Y-P1_Y)*(X_In-P1_X))/(P2_X-P1_X));

END_FUNCTION

// POUs/Utils Functions/LINEAR_BAD
FUNCTION LINEAR_BAD : INT (* Linear interpolation *)
VAR_INPUT
	PuntoMinX	: INT;
	PuntoMaxX	: INT;
	ValIn		: INT;
	PuntoMinY	: REAL;
	PuntoMaxY	: REAL;
	Decimali	: BYTE;
END_VAR
VAR
	Gain				: REAL;
	PuntoMinX_R			: REAL;
	PuntoMaxX_R			: REAL;
	Linearizzazione_R	: REAL;
END_VAR


PuntoMinX_R:=INT_TO_REAL(PuntoMinX);
PuntoMaxX_R:=INT_TO_REAL(PuntoMaxX);

Gain:=(PuntoMaxX_R-PuntoMinX_R)/(PuntoMaxY-PuntoMinY);	(* Calcolo in guadagno per la linarizzazione *)
Linearizzazione_R:=PuntoMinx+(Gain*(ValIn-PuntoMinY));	(* Ottengo il valore linearizzato *)

LINEAR_BAD:=REAL_TO_INT(Linearizzazione_R*(EXPT(10, Decimali)));  (* Ottengo intero con i decimai voluti *)

END_FUNCTION

// POUs/Utils Functions/MEMCLR
FUNCTION MEMCLR:BOOL
VAR_INPUT
	pDestinationAddress:POINTER TO ARRAY[1..2] OF BYTE;
	BytesToClear:WORD;
END_VAR
VAR
END_VAR

WHILE (BytesToClear > 0) DO
	pDestinationAddress^[1]:=0;
	pDestinationAddress:=ADR(pDestinationAddress^[2]); (* increment destination *)
	BytesToClear:=BytesToClear -1; (* decrement number of bytes to copy *)
END_WHILE

END_FUNCTION

// POUs/Plant_Objects/obj_LUXM
FUNCTION_BLOCK obj_LUXM
(* === Metered ON/OFF Illumination Point ===
   Failure detection:
   Statistic data:
   
   - Come identifico l'assenza del nodo?? (Rele non funzionante/non alimentato)
   - Acquisizione carico dopo accensione?? Dati carico in NVM!
   
   v1.0[07/05/15] - Create
*)
VAR_INPUT
	(* Settings *)
	ID				: BYTE;
	(* Controls *)
	CTRL_MODE		: INT:=900;  (* 0:MAN OFF, -1:MAN-ON,
							   -2:KEY-ON, -3:KEY-OFF, -4:DAY, -5:NIGHT,
							   N>0:Nsec-TIMER *)
	CTRL_MODE_backUp: INT;		
	//LuxTimer		: TIME:=T#900S;
	StrLuxTimer		: DWORD:=1500;(* diego: it was 1500 *)
			   
	CTRL_TRIG		: BOOL; (* Trigger for timer start *)
	CTRL_KEY		: BOOL; (* External KEY control input *)
	CTRL_SENS		: BOOL; (* External dark sensor input [1:Dark] *)
	CTRL_EXTON		: BOOL; (* External forced activation *)
	(* Physical inputs *)
	REL_ST			: BOOL; (* Status feedback *)
	REL_V			: WORD; (* [E-1 V] Voltage *)
	REL_A			: WORD; (* [E-1 A] Current *)
	REL_ALM			: WORD; (* Error status [0:OK, 1:Disconnected, 2:LoadLOW, 3:LoadHIGH, 4:Overload, 5:ControlFAIL] *)
	REL_TEMP		: INT;  (* [E-1 °C] Temperature *)
	REL_TON			: DWORD;(* [sec] External working time counter *)  
	(* Persistent *)(*
	WORKINGTIME		: POINTER TO DWORD; (* [sec] Internal working time counter *)
	POWERONCYCLES	: POINTER TO DWORD; (* Internal counter of power-on cycles *)
	ENERGYCOUNTER	: POINTER TO DWORD; (* [E-1 kWh] Internal energy counter *)
	ENERGYCOUNTER_T : POINTER TO DWORD; (* Temporary energy in E-2*Wsec *)*)
	PressKeyVisuMan	: BOOL := 0;
	PressKeyVisuOn	: BOOL := 0;

	TCP_CommandMAN	: bool;
	TCP_CommandON	: bool;
	ModeToServer : byte;
	ForcedOn : byte;
	ForcedOff : byte;	

END_VAR
VAR_IN_OUT
//VAR_OUTPUT RETAIN PERSISTENT
	WORKINGTIME		: DWORD; (* [sec] Internal working time counter *)
	POWERONCYCLES	: DWORD; (* Internal counter of power-on cycles *)
	ENERGYCOUNTER	: DWORD; (* [E-1 kWh] Internal energy counter *)
	ENERGYCOUNTER_T : DWORD; (* Temporary energy in E-2*Wsec *)
END_VAR
VAR_OUTPUT
	(* Physical outputs *)
	REL_EN			: BOOL;	(* Control output *)
	(* Status *)
	Status_Log		: BYTE;
	Status_Vis 		: DWORD;
END_VAR
VAR
	TickTimer		: TON := ( PT:=T#1S );
	TrigTimer		: TOF;
	sREL_EN			: FLT_EVENT;
	sREL_ALM		: WORD:=16#FFFF;
	chkREL_ST		: FLT_TIME := ( TTAP:=T#20S, INITEV:=FALSE );
	
END_VAR

(* Trig timer *)
TrigTimer(IN:=CTRL_TRIG);


(* Control logic *)
IF CTRL_EXTON THEN
	REL_EN:=TRUE;
ELSE
	CASE CTRL_MODE OF
		 0: REL_EN:=FALSE;
		-1: REL_EN:=TRUE;
		-2: REL_EN:=CTRL_KEY;
		-3: REL_EN:=NOT CTRL_KEY;
		-4: REL_EN:=CTRL_SENS;
		-5: REL_EN:=NOT CTRL_SENS;
	ELSE
		IF CTRL_MODE>0 THEN
			REL_EN:=TrigTimer.Q;
			//LuxTimer:=int_to_Time(CTRL_MODE);
			TrigTimer.PT:=T#1S*StrLuxTimer;
			//StrLuxTimer:=Time_to_dword(LuxTimer);
			//StrLuxTimer:=StrLuxTimer/1000;
			//TrigTimer.PT:=T#1S*CTRL_MODE;
		ELSE
			REL_EN:=FALSE;
		END_IF
	END_CASE
END_IF

(* Temporary energy counter *)
TickTimer(IN:=NOT TickTimer.Q);
IF TickTimer.Q AND REL_EN THEN
	WORKINGTIME:=WORKINGTIME+1;
	ENERGYCOUNTER_T:=ENERGYCOUNTER_T+REL_V*REL_A;
	IF ENERGYCOUNTER_T>36000000 THEN
		ENERGYCOUNTER_T:=ENERGYCOUNTER_T-36000000;
		ENERGYCOUNTER:=ENERGYCOUNTER+1;		
	END_IF
END_IF

(* Generate status events *)
sREL_EN(IN:=REL_EN);
IF sREL_EN.EVL THEN LogEv(EL_Log,EO_LUXM,ID,2,''); END_IF
IF sREL_EN.EVH THEN LogEv(EL_Log,EO_LUXM,ID,3,''); POWERONCYCLES:=POWERONCYCLES+1; END_IF

(* Check status feedback *)
chkREL_ST(IN:=(REL_ST<>REL_EN));
IF chkREL_ST.EVH THEN LogEv(EL_Alarm,EO_LUXM,ID,9,''); END_IF
IF chkREL_ST.EVL AND sREL_ALM=0 THEN LogEv(EL_Log,EO_LUXM,ID,1,''); END_IF

(* Check controller alarm *)
IF sREL_ALM<>REL_ALM THEN
	CASE REL_ALM OF
		0: IF NOT chkREL_ST.OUT THEN LogEv(EL_Log,EO_LUXM,ID,1,''); END_IF
		1: LogEv(EL_Alarm,EO_LUXM,ID,6,'');
		2: LogEv(EL_Wrn  ,EO_LUXM,ID,4,WORD_TO_STRING(REL_A));
		3: LogEv(EL_Wrn  ,EO_LUXM,ID,5,WORD_TO_STRING(REL_A));
		4: LogEv(EL_Alarm,EO_LUXM,ID,7,WORD_TO_STRING(REL_A));
		5: LogEv(EL_Alarm,EO_LUXM,ID,8,'');
	END_CASE
	sREL_ALM:=REL_ALM;
END_IF

(* Status color *)
   IF REL_ALM=1 OR REL_ALM>3 OR chkREL_ST.OUT	THEN Status_Log:=2; Status_Vis:=COLOR_RED;
ELSIF REL_ALM<>0								THEN Status_Log:=1; Status_Vis:=COLOR_YELLOW;
                  	   							ELSE Status_Log:=0; Status_Vis:=SEL(REL_EN,COLOR_GREEN_OFF,COLOR_GREEN);
END_IF

ACTION AddLogData:
Logger.s1:=INSERT('&LUX=',BYTE_TO_STRING(ID),4);
IF ID<10 THEN Logger.s1:=INSERT(Logger.s1,'0',4); END_IF
(*
Logger.s1:=CONCAT(Logger.s1,WORD_TO_STRING(REL_V));				Logger.s1:=CONCAT(Logger.s1,';');
Logger.s1:=CONCAT(Logger.s1,WORD_TO_STRING(REL_A));				Logger.s1:=CONCAT(Logger.s1,';');
Logger.s1:=CONCAT(Logger.s1,DWORD_TO_STRING(ENERGYCOUNTER));	Logger.s1:=CONCAT(Logger.s1,';');
Logger.s1:=CONCAT(Logger.s1,DWORD_TO_STRING(WORKINGTIME));		Logger.s1:=CONCAT(Logger.s1,';');
Logger.s1:=CONCAT(Logger.s1,DWORD_TO_STRING(POWERONCYCLES));	Logger.s1:=CONCAT(Logger.s1,';');
Logger.s1:=CONCAT(Logger.s1,INT_TO_STRING(REL_TEMP));			Logger.s1:=CONCAT(Logger.s1,';');

Logger.s1:=CONCAT(Logger.s1,BYTE_TO_STRING(Status_Log));
ADDSTRING(ADR(Logger.TData), ADR(Logger.s1), Logger.TLen);
*)

Logger.s1:=CONCAT(Logger.s1,BOOL_TO_STRING(REL_EN));			Logger.s1:=CONCAT(Logger.s1,';');	
Logger.s1:=CONCAT(Logger.s1,DWORD_TO_STRING(WORKINGTIME));		Logger.s1:=CONCAT(Logger.s1,';');
Logger.s1:=CONCAT(Logger.s1,DWORD_TO_STRING(POWERONCYCLES));	Logger.s1:=CONCAT(Logger.s1,';');

case ModeToServer of
	0: 	// Manuale OFF				
		ModeToServer := 0;
		ForcedOn := 0;
		ForcedOff := 1;
	1:	// Manuale ON				
		ModeToServer := 1;
		ForcedOn := 1;
		ForcedOff := 0;	
	2:	// Cronografo
		ForcedOn := 0;
		ForcedOff := 0;	
	3: //Timer
		ForcedOn := 0;
		ForcedOff := 0;			
end_case

Logger.s1:=CONCAT(Logger.s1,BYTE_TO_STRING(ModeToServer));			Logger.s1:=CONCAT(Logger.s1,';');
Logger.s1:=CONCAT(Logger.s1,BYTE_TO_STRING(Status_Log));			Logger.s1:=CONCAT(Logger.s1,';');
Logger.s1:=CONCAT(Logger.s1,BYTE_TO_STRING(ForcedOn));			Logger.s1:=CONCAT(Logger.s1,';');
Logger.s1:=CONCAT(Logger.s1,BYTE_TO_STRING(ForcedOff));			Logger.s1:=CONCAT(Logger.s1,';');
Logger.s1:=CONCAT(Logger.s1,WORD_TO_STRING(REL_V));				Logger.s1:=CONCAT(Logger.s1,';');
Logger.s1:=CONCAT(Logger.s1,WORD_TO_STRING(REL_A));				Logger.s1:=CONCAT(Logger.s1,';');
Logger.s1:=CONCAT(Logger.s1,DWORD_TO_STRING(ENERGYCOUNTER));	Logger.s1:=CONCAT(Logger.s1,';');
Logger.s1:=CONCAT(Logger.s1,INT_TO_STRING(REL_TEMP));			
ADDSTRING(ADR(Logger.TData), ADR(Logger.s1), Logger.TLen);
END_ACTION

ACTION StatReset:
(* Reset statistic counters *)
WORKINGTIME:=0;
POWERONCYCLES:=0;
ENERGYCOUNTER:=0;
END_ACTION

END_FUNCTION_BLOCK

// POUs/Utils Functions/DELAYRETRY
FUNCTION_BLOCK DELAYRETRY
VAR_INPUT
	RETRIES	: BYTE:=5;
	DELAY	: TIME:=T#5S;
	(*TIMEOUT : TIME:=T#5s; (* Extend to support operation timeout *)*)
END_VAR
VAR_OUTPUT
	RUNNING : BOOL;
	EXEC	: BOOL; (* Execution semaphore *) 
	EV_ERR	: BOOL; (* Retries error *)
	EV_OK	: BOOL; (* Signal recovered state *)
END_VAR
VAR
	retry	: BYTE;
	tm1		: TON;	
END_VAR

EV_ERR:=FALSE;
EV_OK:=FALSE;

IF NOT (RUNNING OR EXEC) THEN
	IF retry=0 THEN EXEC:=TRUE;
	ELSE
		tm1(IN:=TRUE, PT:=DELAY); 
		IF tm1.Q THEN
			EXEC:=TRUE;
		END_IF
	END_IF
END_IF

ACTION Start:
RUNNING:=TRUE;
END_ACTION

ACTION Success:
RUNNING:=FALSE;
IF retry>=RETRIES THEN
	EV_OK:=TRUE;
END_IF
retry:=0;
EXEC:=TRUE;
END_ACTION

ACTION Fail:
RUNNING:=FALSE;
retry:=retry+1;
IF retry=RETRIES THEN
	EV_ERR:=TRUE;
END_IF
EXEC:=FALSE;
tm1(IN:=FALSE);
END_ACTION

END_FUNCTION_BLOCK

// POUs/Utils Functions/RAW16TOHEXSTR
FUNCTION RAW16TOHEXSTR : STRING(128)
VAR_INPUT
	pData: POINTER TO BYTE;
	DataLen: BYTE;
END_VAR
VAR
	pt: POINTER TO BYTE;
	xl: BYTE;
END_VAR

pt:=ADR(RAW16TOHEXSTR);
xl:=0;

WHILE DataLen>0 AND xl<120 DO

	pData:=pData+1;

	pt^ := (pData^ / 16#10) + 48 + (((pData^ / 16#10)/10)*7);
	pt:=pt+1;
	pt^ := (pData^ AND 16#0F)  + 48 + (((pData^ AND 16#0F)/10)*7);
	pt:=pt+1;

	pData:=pData-1;

	pt^ := (pData^ / 16#10) + 48 + (((pData^ / 16#10)/10)*7);
	pt:=pt+1;
	pt^ := (pData^ AND 16#0F)  + 48 + (((pData^ AND 16#0F)/10)*7);
	pt:=pt+1;

	xl:=xl+4;

	DataLen:=DataLen-2;
	pData:=pData+2;

END_WHILE

pt^:=0;

END_FUNCTION

// POUs/Utils Functions/RAWTOHEXSTR
FUNCTION RAWTOHEXSTR : STRING(128)
VAR_INPUT
	pData: POINTER TO BYTE;
	DataLen: BYTE;
END_VAR
VAR
	pt: POINTER TO BYTE;
	xl: BYTE;
END_VAR

pt:=ADR(RAWTOHEXSTR);

xl:=2;

WHILE DataLen>0 AND xl<128 DO

	pt^ := (pData^ / 16#10) + 48 + (((pData^ / 16#10)/10)*7);
	pt:=pt+1;
	pt^ := (pData^ AND 16#0F)  + 48 + (((pData^ AND 16#0F)/10)*7);
	pt:=pt+1;

	xl:=xl+2;

	DataLen:=DataLen-1;
	pData:=pData+1;

END_WHILE

pt^:=0;

END_FUNCTION

// POUs/Utils Functions/TONOF
FUNCTION_BLOCK TONOF
VAR_INPUT
	IN		: BOOL;
	PT_ON	: TIME; (* time to pass, before OUT is set *)
	PT_OF	: TIME; (* time to pass, before OUT is reset *)
END_VAR
VAR_OUTPUT
	OUT		: BOOL;
END_VAR
VAR
	timer	: TON;
END_VAR

IF IN<>OUT THEN
	timer(IN:=TRUE,PT:=SEL(IN,PT_OF,PT_ON));
	IF timer.Q THEN OUT:=IN; END_IF
ELSE
	timer(IN:=FALSE);
END_IF

END_FUNCTION_BLOCK

// POUs/Plant_Objects/obj_ZREL
FUNCTION_BLOCK obj_ZREL
(* === ZIGBEE CONTROL RELE REL-100 ===
   v1.0[07/05/05] - Create
*)
VAR_INPUT
	(* Settings *)
	ID				: BYTE;
	ADDRESS			: BYTE;
	ADDRESSGW		: BYTE:=0;
	Refresh_Period	: TIME:=t#3m;
	(* Controls *)
	REL_CTRL		: BOOL;
	Refresh_Auto	: BOOL:=TRUE; (* Enable automatic refresh *)
	Refresh_Now		: BOOL; 	  (* Force an immediate refresh *)
	Request_Learn	: BOOL;		  (* Request load learning *)
END_VAR
VAR_IN_OUT
	(* Interface *)
	MODBUS			: obj_MODBUS_TCP;
END_VAR
VAR_OUTPUT
	(* Load status *)
	ONLINE			: BOOL; (* Network presence *)
	REL_ST			: BOOL; (* Status feedback *)
	REL_V			: WORD; (* [E-1 V] Voltage *)
	REL_A			: WORD; (* [E-1 A] Current *)
	REL_ALM			: WORD; (* Error status [0:OK, 1:Disconnected, 2:LoadLOW, 3:LoadHIGH, 4:Overload, 5:ControlFAIL] *)
	REL_TEMP		: INT;  (* [E-1 °C] Temperature *)
	REL_LQI			: BYTE;
	REL_TON			: DWORD;(* [sec] Working time counter *)  
	(* Status *)
	Status_Log		: BYTE:=1;
	Status_Vis 		: DWORD:=COLOR_LBLUE;
END_VAR
VAR CONSTANT
	ST_UNKNOWN		: BYTE:=0;
	ST_WAITPRESENCE	: BYTE:=1;
	ST_SETUP1		: BYTE:=2;
	ST_SETUP2		: BYTE:=3;
	ST_SETUP3		: BYTE:=4;
	ST_SETVAR		: BYTE:=6;
	ST_RUN			: BYTE:=10;
	ST_STATUS1		: BYTE:=20;
	ST_STATUS2		: BYTE:=21;
	ST_LEARN1		: BYTE:=30;
END_VAR
VAR
	dtry		: DELAYRETRY;
	stm			: BYTE:=0;
	dly 	 	: TON := (PT:=T#5S);
	dlyctrl		: TON := (PT:=T#5S);
	outw		: WORD;
	bus_st0		: WORD:=0;
	
END_VAR

outw:=BOOL_TO_WORD(REL_CTRL);

(* Auto refresh timer *)
dlyctrl(IN:=NOT (dlyctrl.Q OR (REL_CTRL=REL_ST)));
dly(IN:=NOT (dly.Q OR Refresh_Now OR (NOT Refresh_Auto)));
IF dly.Q OR dlyctrl.Q THEN dly.PT:=Refresh_Period; Refresh_Now:=TRUE; END_IF

ZREL_STATUS_ALIGNED[ID]:=(REL_CTRL=REL_ST);


(* Stm *)
dtry();
CASE stm OF
	
	ST_UNKNOWN:
		stm:=ST_SETVAR;  //GIURE ver 02test
		return;  //GIURE ver 02test	
		(* Request node status *)
		IF dtry.EXEC AND MODBUS.MB_Ready AND NOT MODBUS.MB_Lock THEN
			dtry.Start();
			MODBUS.MB_Lock:=TRUE;
			MB_Req_NetStatus();
			stm:=ST_WAITPRESENCE;
		END_IF

	ST_WAITPRESENCE:
		(* Wait node status response *)
		IF NOT MODBUS.MB_Start THEN
			MB_Response();
			IF bus_St0=0 AND MODBUS.MB_READBUF[0]<>3 THEN
				dtry.Success();
				IF dtry.EV_OK THEN LogEv(EL_Log,EO_ZREL,ID,1,'Online');	END_IF
//				MB_Set_DefaultMode(); //GIURE ver 02test
				stm:=ST_SETUP1; 
			ELSE
				dtry.Fail();
				IF dtry.EV_ERR AND Status_Log<>2 THEN
					Status_Log:=2; Status_Vis:=COLOR_RED;
					LogEv(EL_Alarm,EO_ZREL,ID,2,'Offline');
				END_IF
				MODBUS.MB_Lock:=FALSE;
				stm:=ST_UNKNOWN;
			END_IF
		END_IF

	ST_SETUP1:
		IF NOT MODBUS.MB_Start THEN
			MB_Response();
			IF bus_st0>0 THEN MODBUS.MB_Lock:=FALSE; stm:=ST_UNKNOWN;
						 //ELSE MB_Set_DefaultMode(); stm:=ST_SETUP2;	 //GIURE ver 02test				
			END_IF
		END_IF

	ST_SETUP2:
		IF NOT MODBUS.MB_Start THEN
			MB_Response();
			IF bus_st0>0 THEN MODBUS.MB_Lock:=FALSE; stm:=ST_UNKNOWN;
						// ELSE MB_Set_DefaultMode(); stm:=ST_SETUP3;  //GIURE ver 02test
			END_IF
		END_IF

	ST_SETUP3:
		IF NOT MODBUS.MB_Start THEN
			MB_Response();
			IF bus_st0>0 THEN MODBUS.MB_Lock:=FALSE; stm:=ST_UNKNOWN;
						// ELSE MB_Set_DefaultMode(); stm:=ST_SETVAR; //GIURE ver 02test
		 END_IF
		END_IF

	ST_SETVAR:
		(* Initialize var manager *)
		IF NOT MODBUS.MB_Start THEN
			MB_Response();
			MODBUS.MB_Lock:=0;
			IF bus_st0>0 THEN stm:=ST_UNKNOWN;
			ELSE
				MODBUS.VAR_Pointer:=ADR(outw);
				MODBUS.VAR_Search();
				MODBUS.VAR_Cfg^.Variable      :=MODBUS.VAR_Pointer;
				MODBUS.VAR_Cfg^.Variable_Size :=1;
				MODBUS.VAR_Cfg^.SlaveAddress  :=ADDRESS;
				MODBUS.VAR_Cfg^.FunCode       :=6;
				MODBUS.VAR_Cfg^.FunAddress    :=319;		//probabile errore!!! il registro a cui settare il timer è il successivo 320 (registro 321)
				MODBUS.VAR_Cfg^.Refresh_Time  :=120+ID;		//Valore che indica la durata del test utile per l'autoapprendimento dei valori di consumo standard
				MODBUS.VARS_En:=TRUE;
				stm:=ST_RUN;
			END_IF
		END_IF
		
	ST_RUN: (* Runtime *)
		IF Refresh_Now AND NOT MODBUS.MB_Lock THEN
			Refresh_Now:=FALSE;
			MODBUS.MB_Lock:=TRUE;
			MB_Req_NetStatus();
			stm:=ST_STATUS1;
		END_IF
		IF Request_Learn AND NOT MODBUS.MB_Lock THEN
			Request_Learn:=FALSE;
			MODBUS.MB_Lock:=TRUE;
			MB_Set_AutoLearn();
			stm:=ST_LEARN1;
		END_IF
		(* Check status *)
		IF Status_Log<>0 AND REL_LQI>=100 AND REL_ALM<>5 AND ONLINE THEN	//AND REL_LQI>=100 giure
			LogEv(EL_Alarm,EO_ZREL,ID,1,''); Status_Log:=0;
		END_IF
		IF Status_Log<2 THEN
			IF NOT ONLINE THEN
				LogEv(EL_Alarm,EO_ZREL,ID,3,''); Status_Log:=2; Status_Vis:=COLOR_RED;
			ELSIF REL_ALM=5 THEN
				LogEv(EL_Alarm,EO_ZREL,ID,6,''); Status_Log:=2; Status_Vis:=COLOR_RED;
			END_IF
		END_IF
		IF Status_Log=0 THEN
			IF REL_LQI<100 THEN
				LogEv(EL_Alarm,EO_ZREL,ID,2,BYTE_TO_STRING(REL_LQI)); Status_Log:=1; Status_Vis:=COLOR_YELLOW;
			ELSIF REL_TEMP<-50 OR REL_TEMP>800 THEN
				LogEv(EL_Alarm,EO_ZREL,ID,5,INT_TO_STRING(REL_TEMP)); Status_Log:=1; Status_Vis:=COLOR_YELLOW;
			ELSE
				Status_Vis:=SEL(REL_ST,COLOR_GREEN_OFF,COLOR_GREEN);
			END_IF
		END_IF

	ST_STATUS1:
		IF NOT MODBUS.MB_Start THEN
			MB_Response();
			IF bus_st0=0 THEN
				(* Read net status data *)
				ONLINE:=(MODBUS.MB_READBUF[0]<>3);
			END_IF
			MB_Req_Status();
			stm:=ST_STATUS2;
		END_IF

	ST_STATUS2:
		IF NOT MODBUS.MB_Start THEN
			MB_Response();
			IF bus_st0=0 THEN
				(* Read status data *)
				REL_ST  :=MODBUS.MB_READBUF[0]<>0;
				REL_V   :=2300;	//MODBUS.MB_READBUF[1];
				REL_A   :=20;	//MODBUS.MB_READBUF[2];
				REL_ALM :=0;	//MODBUS.MB_READBUF[3];
				REL_LQI :=250;	//WORD_TO_BYTE(MODBUS.MB_READBUF[4]); GIURE
				REL_TEMP:=250; //ADR_AT_INT(ADR(MODBUS.MB_READBUF[5]));
				REL_TON :=16#10000*MODBUS.MB_READBUF[6]+MODBUS.MB_READBUF[7];
			END_IF
			MODBUS.MB_Lock:=FALSE;
			stm:=ST_RUN;
		END_IF

	ST_LEARN1: (* Configuration response 1 *)
		IF NOT MODBUS.MB_Start THEN
			MB_Response();
			MODBUS.MB_Lock:=FALSE;
			stm:=ST_RUN;
		END_IF
	
END_CASE

ACTION AddLogData:
Logger.s1:=INSERT('&ZREL=',BYTE_TO_STRING(ID),5);
IF ID<10 THEN Logger.s1:=INSERT(Logger.s1,'0',5); END_IF

Logger.s1:=CONCAT(Logger.s1,INT_TO_STRING(REL_TEMP));		Logger.s1:=CONCAT(Logger.s1,';');
Logger.s1:=CONCAT(Logger.s1,'0');							Logger.s1:=CONCAT(Logger.s1,';');
Logger.s1:=CONCAT(Logger.s1,BYTE_TO_STRING(REL_LQI));		Logger.s1:=CONCAT(Logger.s1,';');

Logger.s1:=CONCAT(Logger.s1,BYTE_TO_STRING(Status_Log));
ADDSTRING(ADR(Logger.TData), ADR(Logger.s1), Logger.TLen);
END_ACTION

ACTION MB_Req_NetStatus:
MODBUS.MB_MASTER.bUNIT_ID        :=ADDRESSGW;
MODBUS.MB_MASTER.bFUNCTION_CODE  :=3;
MODBUS.MB_MASTER.wREAD_ADDRESS   :=13;
MODBUS.MB_MASTER.wREAD_QUANTITY  :=1;
MODBUS.MB_MASTER.wWRITE_ADDRESS  :=0;
MODBUS.MB_MASTER.wWRITE_QUANTITY :=0;
MODBUS.MB_Start:=TRUE;
END_ACTION

ACTION MB_Set_DefaultMode:
(*
	 331(Offline mode)    :=2(always on)
	 332(Offline timeout) :=240+ID
	 333(Poweron mode)    :=1(always on)
	 334(Operating mode)  :=0(manual)
*)
(*MODBUS.MB_MASTER.bUNIT_ID        :=ADDRESS;
MODBUS.MB_MASTER.bFUNCTION_CODE  :=16;
MODBUS.MB_MASTER.wREAD_ADDRESS   :=0;
MODBUS.MB_MASTER.wREAD_QUANTITY  :=0;
MODBUS.MB_MASTER.wWRITE_ADDRESS  :=331; 
MODBUS.MB_MASTER.wWRITE_QUANTITY :=4;
MODBUS.MB_WRITEBUF[0]:=2;
MODBUS.MB_WRITEBUF[1]:=250+ID;
MODBUS.MB_WRITEBUF[2]:=1;
MODBUS.MB_WRITEBUF[3]:=0;
MODBUS.MB_Start:=TRUE;*)

CASE stm OF
	
	ST_WAITPRESENCE:	//scrittura nel registro 332 l'impostazione 2 ovvero: acceso se offline
		MODBUS.MB_MASTER.bUNIT_ID        :=ADDRESS;
		MODBUS.MB_MASTER.bFUNCTION_CODE  :=6;
		MODBUS.MB_MASTER.wREAD_ADDRESS   :=0;
		MODBUS.MB_MASTER.wREAD_QUANTITY  :=0;
		MODBUS.MB_MASTER.wWRITE_ADDRESS  :=331; 
		MODBUS.MB_MASTER.wWRITE_QUANTITY :=1;
		MODBUS.MB_WRITEBUF[0]:=2;	//on if offline
		MODBUS.MB_Start:=TRUE;

	ST_SETUP1:	//set del timeout al valore 250+ID (registro 333)
		MODBUS.MB_MASTER.wWRITE_ADDRESS	:=332;
		MODBUS.MB_WRITEBUF[0]:=250+ID;
		MODBUS.MB_Start:=TRUE;

	ST_SETUP2: //set del modo di funzionamento all'accensione (registro 334) (0=always off (default), 1=always on, 2=with timer)
		MODBUS.MB_MASTER.wWRITE_ADDRESS	:=333;
		MODBUS.MB_WRITEBUF[0]:=1;
		MODBUS.MB_Start:=TRUE;

	ST_SETUP3://set del modo di funzionamento generale(registro 335) (0=on request (default), 1=with timer)
		MODBUS.MB_MASTER.wWRITE_ADDRESS	:=334;
		MODBUS.MB_WRITEBUF[0]:=0;
		MODBUS.MB_Start:=TRUE;

END_CASE
END_ACTION

ACTION MB_Req_Status:
MODBUS.MB_MASTER.bUNIT_ID        :=ADDRESS;
MODBUS.MB_MASTER.bFUNCTION_CODE  :=3;
MODBUS.MB_MASTER.wREAD_ADDRESS   :=300;
MODBUS.MB_MASTER.wREAD_QUANTITY  :=8;
MODBUS.MB_MASTER.wWRITE_ADDRESS  :=0;
MODBUS.MB_MASTER.wWRITE_QUANTITY :=0;
MODBUS.MB_Start:=TRUE;
END_ACTION

ACTION MB_Set_AutoLearn:
MODBUS.MB_MASTER.bUNIT_ID        :=ADDRESS;
MODBUS.MB_MASTER.bFUNCTION_CODE  :=6;
MODBUS.MB_MASTER.wREAD_ADDRESS   :=0;
MODBUS.MB_MASTER.wREAD_QUANTITY  :=0;
MODBUS.MB_MASTER.wWRITE_ADDRESS  :=321;
MODBUS.MB_MASTER.wWRITE_QUANTITY :=1;
MODBUS.MB_WRITEBUF[0]:=2;
MODBUS.MB_Start:=TRUE;
END_ACTION

ACTION MB_Response:
IF bus_st0<>MODBUS.MB_MASTER.wERROR THEN
	bus_st0:=MODBUS.MB_MASTER.wERROR;
	IF bus_st0<>0 THEN
		LogEv(EL_Alarm,EO_ZREL,ID,4,WORD_TO_STRING(bus_st0));
	END_IF
END_IF
END_ACTION

END_FUNCTION_BLOCK

// POUs/Utils Functions/ADR_AT_INT
FUNCTION ADR_AT_INT : INT
VAR_INPUT
	ADDRESS : POINTER TO INT;
END_VAR
VAR
END_VAR

ADR_AT_INT:=ADDRESS^;

END_FUNCTION

